          SLIN XP129 WITH $VEL = SVEL_CP(0.1, , LCPDAT33), $TOOL = STOOL2(FP129), $BASE = SBASE(FP129.BASE_NO), $IPO_MODE = SIPO_MODE(FP129.IPO_FRAME), $LOAD = SLOAD(FP129.TOOL_NO), $ACC = SACC_CP(LCPDAT33), $ORI_TYPE = SORI_TYP(LCPDAT33), $APO = SAPO(LCPDAT33), $JERK = SJERK(LCPDAT33), $COLLMON_TOL_PRO[1] = USE_CM_PRO_VALUES(0)
          ;ENDFOLD
          ;FOLD SPTP P500 Vel=100 % PDAT19 Tool[1]:SMC Base[0] ;%{PE}
          ;FOLD Parameters ;%{h}
          ;Params IlfProvider=kukaroboter.basistech.inlineforms.movement.spline; Kuka.IsGlobalPoint=False; Kuka.PointName=P500; Kuka.BlendingEnabled=False; Kuka.MoveDataPtpName=PDAT19; Kuka.VelocityPtp=100; Kuka.VelocityFieldEnabled=True; Kuka.ColDetectFieldEnabled=True; Kuka.CurrentCDSetIndex=0; Kuka.MovementParameterFieldEnabled=True; IlfCommand=SPTP
          ;ENDFOLD
          SPTP XP500 WITH $VEL_AXIS[1] = SVEL_JOINT(100.0), $TOOL = STOOL2(FP500), $BASE = SBASE(FP500.BASE_NO), $IPO_MODE = SIPO_MODE(FP500.IPO_FRAME), $LOAD = SLOAD(FP500.TOOL_NO), $ACC_AXIS[1] = SACC_JOINT(PPDAT19), $APO = SAPO_PTP(PPDAT19), $GEAR_JERK[1] = SGEAR_JERK(PPDAT19), $COLLMON_TOL_PRO[1] = USE_CM_PRO_VALUES(0)
          ;ENDFOLD
          ;FOLD Gripper SET [1]Gripper1 State=[1]ABIERTA Wait 0.2[s] Check with Strategy 1 ;%{PE}
          ;FOLD Parameters Parameters ;%{h}
          ;Params IlfProvider=GripperTech.GripperSet;setgripper=1;setstate=1;setcont=nocont;waittime=0.2;errorstrategy=1
          ;ENDFOLD
          GRPg_SetStateAndCheck(1, 1, 0.2, 1)
          ;ENDFOLD
      ENDIF
      IF eatPosition == 30 THEN
          ;FOLD SPTP P130 Vel=100 % PDAT1 Tool[1]:SMC Base[0] ;%{PE}
          ;FOLD Parameters ;%{h}
          ;Params IlfProvider=kukaroboter.basistech.inlineforms.movement.spline; Kuka.IsGlobalPoint=False; Kuka.PointName=P130; Kuka.BlendingEnabled=False; Kuka.MoveDataPtpName=PDAT1; Kuka.VelocityPtp=100; Kuka.VelocityFieldEnabled=True; Kuka.ColDetectFieldEnabled=True; Kuka.CurrentCDSetIndex=0; Kuka.MovementParameterFieldEnabled=True; IlfCommand=SPTP
          ;ENDFOLD
          SPTP XP130 WITH $VEL_AXIS[1] = SVEL_JOINT(100.0), $TOOL = STOOL2(FP130), $BASE = SBASE(FP130.BASE_NO), $IPO_MODE = SIPO_MODE(FP130.IPO_FRAME), $LOAD = SLOAD(FP130.TOOL_NO), $ACC_AXIS[1] = SACC_JOINT(PPDAT1), $APO = SAPO_PTP(PPDAT1), $GEAR_JERK[1] = SGEAR_JERK(PPDAT1), $COLLMON_TOL_PRO[1] = USE_CM_PRO_VALUES(0)
          ;ENDFOLD
          ;FOLD SLIN P230 Vel=0.1 m/s CPDAT32 Tool[1]:SMC Base[0] ;%{PE}
          ;FOLD Parameters ;%{h}
          ;Params IlfProvider=kukaroboter.basistech.inlineforms.movement.spline; Kuka.IsGlobalPoint=False; Kuka.PointName=P230; Kuka.BlendingEnabled=False; Kuka.MoveDataName=CPDAT32; Kuka.VelocityPath=0.1; Kuka.VelocityFieldEnabled=True; Kuka.ColDetectFieldEnabled=True; Kuka.CurrentCDSetIndex=0; Kuka.MovementParameterFieldEnabled=True; IlfCommand=SLIN
          ;ENDFOLD
          SLIN XP230 WITH $VEL = SVEL_CP(0.1, , LCPDAT32), $TOOL = STOOL2(FP230), $BASE = SBASE(FP230.BASE_NO), $IPO_MODE = SIPO_MODE(FP230.IPO_FRAME), $LOAD = SLOAD(FP230.TOOL_NO), $ACC = SACC_CP(LCPDAT32), $ORI_TYPE = SORI_TYP(LCPDAT32), $APO = SAPO(LCPDAT32), $JERK = SJERK(LCPDAT32), $COLLMON_TOL_PRO[1] = USE_CM_PRO_VALUES(0)
          ;ENDFOLD
          ;FOLD Gripper SET [1]Gripper1 State=[2]CERRADA Wait 0.2[s] Check with Strategy 1 ;%{PE}
          ;FOLD Parameters Parameters ;%{h}
          ;Params IlfProvider=GripperTech.GripperSet;setgripper=1;setstate=2;setcont=nocont;waittime=0.2;errorstrategy=1
          ;ENDFOLD
          GRPg_SetStateAndCheck(1, 2, 0.2, 1)
          ;ENDFOLDinitialPosition
          ;FOLD SLIN P130 Vel=0.1 m/s CPDAT33 Tool[1]:SMC Base[0] ;%{PE}
          ;FOLD Parameters ;%{h}s
          ;Params IlfProvider=kukaroboter.basistech.inlineforms.movement.spline; Kuka.IsGlobalPoint=False; Kuka.PointName=P130; Kuka.BlendingEnabled=False; Kuka.MoveDataName=CPDAT33; Kuka.VelocityPath=0.1; Kuka.VelocityFieldEnabled=True; Kuka.ColDetectFieldEnabled=True; Kuka.CurrentCDSetIndex=0; Kuka.MovementParameterFieldEnabled=True; IlfCommand=SLIN
          ;ENDFOLD
          SLIN XP130 WITH $VEL = SVEL_CP(0.1, , LCPDAT33), $TOOL = STOOL2(FP130), $BASE = SBASE(FP130.BASE_NO), $IPO_MODE = SIPO_MODE(FP130.IPO_FRAME), $LOAD = SLOAD(FP130.TOOL_NO), $ACC = SACC_CP(LCPDAT33), $ORI_TYPE = SORI_TYP(LCPDAT33), $APO = SAPO(LCPDAT33), $JERK = SJERK(LCPDAT33), $COLLMON_TOL_PRO[1] = USE_CM_PRO_VALUES(0)
          ;ENDFOLD
          ;FOLD SPTP P500 Vel=100 % PDAT19 Tool[1]:SMC Base[0] ;%{PE}
          ;FOLD Parameters ;%{h}
          ;Params IlfProvider=kukaroboter.basistech.inlineforms.movement.spline; Kuka.IsGlobalPoint=False; Kuka.PointName=P500; Kuka.BlendingEnabled=False; Kuka.MoveDataPtpName=PDAT19; Kuka.VelocityPtp=100; Kuka.VelocityFieldEnabled=True; Kuka.ColDetectFieldEnabled=True; Kuka.CurrentCDSetIndex=0; Kuka.MovementParameterFieldEnabled=True; IlfCommand=SPTP
          ;ENDFOLD
          SPTP XP500 WITH $VEL_AXIS[1] = SVEL_JOINT(100.0), $TOOL = STOOL2(FP500), $BASE = SBASE(FP500.BASE_NO), $IPO_MODE = SIPO_MODE(FP500.IPO_FRAME), $LOAD = SLOAD(FP500.TOOL_NO), $ACC_AXIS[1] = SACC_JOINT(PPDAT19), $APO = SAPO_PTP(PPDAT19), $GEAR_JERK[1] = SGEAR_JERK(PPDAT19), $COLLMON_TOL_PRO[1] = USE_CM_PRO_VALUES(0)
          ;ENDFOLD
          ;FOLD Gripper SET [1]Gripper1 State=[1]ABIERTA Wait 0.2[s] Check with Strategy 1 ;%{PE}
          ;FOLD Parameters Parameters ;%{h}
          ;Params IlfProvider=GripperTech.GripperSet;setgripper=1;setstate=1;setcont=nocont;waittime=0.2;errorstrategy=1
          ;ENDFOLD
          GRPg_SetStateAndCheck(1, 1, 0.2, 1)
          ;ENDFOLD
      ENDIF
      IF eatPosition == 31 THEN
          ;FOLD SPTP P131 Vel=100 % PDAT1 Tool[1]:SMC Base[0] ;%{PE}
          ;FOLD Parameters ;%{h}
          ;Params IlfProvider=kukaroboter.basistech.inlineforms.movement.spline; Kuka.IsGlobalPoint=False; Kuka.PointName=P131; Kuka.BlendingEnabled=False; Kuka.MoveDataPtpName=PDAT1; Kuka.VelocityPtp=100; Kuka.VelocityFieldEnabled=True; Kuka.ColDetectFieldEnabled=True; Kuka.CurrentCDSetIndex=0; Kuka.MovementParameterFieldEnabled=True; IlfCommand=SPTP
          ;ENDFOLD
          SPTP XP131 WITH $VEL_AXIS[1] = SVEL_JOINT(100.0), $TOOL = STOOL2(FP131), $BASE = SBASE(FP131.BASE_NO), $IPO_MODE = SIPO_MODE(FP131.IPO_FRAME), $LOAD = SLOAD(FP131.TOOL_NO), $ACC_AXIS[1] = SACC_JOINT(PPDAT1), $APO = SAPO_PTP(PPDAT1), $GEAR_JERK[1] = SGEAR_JERK(PPDAT1), $COLLMON_TOL_PRO[1] = USE_CM_PRO_VALUES(0)
          ;ENDFOLD
          ;FOLD SLIN P231 Vel=0.1 m/s CPDAT32 Tool[1]:SMC Base[0] ;%{PE}
          ;FOLD Parameters ;%{h}
          ;Params IlfProvider=kukaroboter.basistech.inlineforms.movement.spline; Kuka.IsGlobalPoint=False; Kuka.PointName=P231; Kuka.BlendingEnabled=False; Kuka.MoveDataName=CPDAT32; Kuka.VelocityPath=0.1; Kuka.VelocityFieldEnabled=True; Kuka.ColDetectFieldEnabled=True; Kuka.CurrentCDSetIndex=0; Kuka.MovementParameterFieldEnabled=True; IlfCommand=SLIN
          ;ENDFOLD
          SLIN XP231 WITH $VEL = SVEL_CP(0.1, , LCPDAT32), $TOOL = STOOL2(FP231), $BASE = SBASE(FP231.BASE_NO), $IPO_MODE = SIPO_MODE(FP231.IPO_FRAME), $LOAD = SLOAD(FP231.TOOL_NO), $ACC = SACC_CP(LCPDAT32), $ORI_TYPE = SORI_TYP(LCPDAT32), $APO = SAPO(LCPDAT32), $JERK = SJERK(LCPDAT32), $COLLMON_TOL_PRO[1] = USE_CM_PRO_VALUES(0)
          ;ENDFOLD
          ;FOLD Gripper SET [1]Gripper1 State=[2]CERRADA Wait 0.2[s] Check with Strategy 1 ;%{PE}
          ;FOLD Parameters Parameters ;%{h}
          ;Params IlfProvider=GripperTech.GripperSet;setgripper=1;setstate=2;setcont=nocont;waittime=0.2;errorstrategy=1
          ;ENDFOLD
          GRPg_SetStateAndCheck(1, 2, 0.2, 1)
          ;ENDFOLDinitialPosition
          ;FOLD SLIN P131 Vel=0.1 m/s CPDAT33 Tool[1]:SMC Base[0] ;%{PE}
          ;FOLD Parameters ;%{h}s
          ;Params IlfProvider=kukaroboter.basistech.inlineforms.movement.spline; Kuka.IsGlobalPoint=False; Kuka.PointName=P131; Kuka.BlendingEnabled=False; Kuka.MoveDataName=CPDAT33; Kuka.VelocityPath=0.1; Kuka.VelocityFieldEnabled=True; Kuka.ColDetectFieldEnabled=True; Kuka.CurrentCDSetIndex=0; Kuka.MovementParameterFieldEnabled=True; IlfCommand=SLIN
          ;ENDFOLD
          SLIN XP131 WITH $VEL = SVEL_CP(0.1, , LCPDAT33), $TOOL = STOOL2(FP131), $BASE = SBASE(FP131.BASE_NO), $IPO_MODE = SIPO_MODE(FP131.IPO_FRAME), $LOAD = SLOAD(FP131.TOOL_NO), $ACC = SACC_CP(LCPDAT33), $ORI_TYPE = SORI_TYP(LCPDAT33), $APO = SAPO(LCPDAT33), $JERK = SJERK(LCPDAT33), $COLLMON_TOL_PRO[1] = USE_CM_PRO_VALUES(0)
          ;ENDFOLD
          ;FOLD SPTP P500 Vel=100 % PDAT19 Tool[1]:SMC Base[0] ;%{PE}
          ;FOLD Parameters ;%{h}
          ;Params IlfProvider=kukaroboter.basistech.inlineforms.movement.spline; Kuka.IsGlobalPoint=False; Kuka.PointName=P500; Kuka.BlendingEnabled=False; Kuka.MoveDataPtpName=PDAT19; Kuka.VelocityPtp=100; Kuka.VelocityFieldEnabled=True; Kuka.ColDetectFieldEnabled=True; Kuka.CurrentCDSetIndex=0; Kuka.MovementParameterFieldEnabled=True; IlfCommand=SPTP
          ;ENDFOLD
          SPTP XP500 WITH $VEL_AXIS[1] = SVEL_JOINT(100.0), $TOOL = STOOL2(FP500), $BASE = SBASE(FP500.BASE_NO), $IPO_MODE = SIPO_MODE(FP500.IPO_FRAME), $LOAD = SLOAD(FP500.TOOL_NO), $ACC_AXIS[1] = SACC_JOINT(PPDAT19), $APO = SAPO_PTP(PPDAT19), $GEAR_JERK[1] = SGEAR_JERK(PPDAT19), $COLLMON_TOL_PRO[1] = USE_CM_PRO_VALUES(0)
          ;ENDFOLD
          ;FOLD Gripper SET [1]Gripper1 State=[1]ABIERTA Wait 0.2[s] Check with Strategy 1 ;%{PE}
          ;FOLD Parameters Parameters ;%{h}
          ;Params IlfProvider=GripperTech.GripperSet;setgripper=1;setstate=1;setcont=nocont;waittime=0.2;errorstrategy=1
          ;ENDFOLD
          GRPg_SetStateAndCheck(1, 1, 0.2, 1)
          ;ENDFOLD
      ENDIF
      IF eatPosition == 32 THEN
          ;FOLD SPTP P132 Vel=100 % PDAT1 Tool[1]:SMC Base[0] ;%{PE}
          ;FOLD Parameters ;%{h}
          ;Params IlfProvider=kukaroboter.basistech.inlineforms.movement.spline; Kuka.IsGlobalPoint=False; Kuka.PointName=P132; Kuka.BlendingEnabled=False; Kuka.MoveDataPtpName=PDAT1; Kuka.VelocityPtp=100; Kuka.VelocityFieldEnabled=True; Kuka.ColDetectFieldEnabled=True; Kuka.CurrentCDSetIndex=0; Kuka.MovementParameterFieldEnabled=True; IlfCommand=SPTP
          ;ENDFOLD
          SPTP XP132 WITH $VEL_AXIS[1] = SVEL_JOINT(100.0), $TOOL = STOOL2(FP132), $BASE = SBASE(FP132.BASE_NO), $IPO_MODE = SIPO_MODE(FP132.IPO_FRAME), $LOAD = SLOAD(FP132.TOOL_NO), $ACC_AXIS[1] = SACC_JOINT(PPDAT1), $APO = SAPO_PTP(PPDAT1), $GEAR_JERK[1] = SGEAR_JERK(PPDAT1), $COLLMON_TOL_PRO[1] = USE_CM_PRO_VALUES(0)
          ;ENDFOLD
          ;FOLD SLIN P232 Vel=0.1 m/s CPDAT32 Tool[1]:SMC Base[0] ;%{PE}
          ;FOLD Parameters ;%{h}
          ;Params IlfProvider=kukaroboter.basistech.inlineforms.movement.spline; Kuka.IsGlobalPoint=False; Kuka.PointName=P232; Kuka.BlendingEnabled=False; Kuka.MoveDataName=CPDAT32; Kuka.VelocityPath=0.1; Kuka.VelocityFieldEnabled=True; Kuka.ColDetectFieldEnabled=True; Kuka.CurrentCDSetIndex=0; Kuka.MovementParameterFieldEnabled=True; IlfCommand=SLIN
          ;ENDFOLD
          SLIN XP232 WITH $VEL = SVEL_CP(0.1, , LCPDAT32), $TOOL = STOOL2(FP232), $BASE = SBASE(FP232.BASE_NO), $IPO_MODE = SIPO_MODE(FP232.IPO_FRAME), $LOAD = SLOAD(FP232.TOOL_NO), $ACC = SACC_CP(LCPDAT32), $ORI_TYPE = SORI_TYP(LCPDAT32), $APO = SAPO(LCPDAT32), $JERK = SJERK(LCPDAT32), $COLLMON_TOL_PRO[1] = USE_CM_PRO_VALUES(0)
          ;ENDFOLD
          ;FOLD Gripper SET [1]Gripper1 State=[2]CERRADA Wait 0.2[s] Check with Strategy 1 ;%{PE}
          ;FOLD Parameters Parameters ;%{h}
          ;Params IlfProvider=GripperTech.GripperSet;setgripper=1;setstate=2;setcont=nocont;waittime=0.2;errorstrategy=1
          ;ENDFOLD
          GRPg_SetStateAndCheck(1, 2, 0.2, 1)
          ;ENDFOLDinitialPosition
          ;FOLD SLIN P132 Vel=0.1 m/s CPDAT33 Tool[1]:SMC Base[0] ;%{PE}
          ;FOLD Parameters ;%{h}s
          ;Params IlfProvider=kukaroboter.basistech.inlineforms.movement.spline; Kuka.IsGlobalPoint=False; Kuka.PointName=P132; Kuka.BlendingEnabled=False; Kuka.MoveDataName=CPDAT33; Kuka.VelocityPath=0.1; Kuka.VelocityFieldEnabled=True; Kuka.ColDetectFieldEnabled=True; Kuka.CurrentCDSetIndex=0; Kuka.MovementParameterFieldEnabled=True; IlfCommand=SLIN
          ;ENDFOLD
          SLIN XP132 WITH $VEL = SVEL_CP(0.1, , LCPDAT33), $TOOL = STOOL2(FP132), $BASE = SBASE(FP132.BASE_NO), $IPO_MODE = SIPO_MODE(FP132.IPO_FRAME), $LOAD = SLOAD(FP132.TOOL_NO), $ACC = SACC_CP(LCPDAT33), $ORI_TYPE = SORI_TYP(LCPDAT33), $APO = SAPO(LCPDAT33), $JERK = SJERK(LCPDAT33), $COLLMON_TOL_PRO[1] = USE_CM_PRO_VALUES(0)
          ;ENDFOLD
          ;FOLD SPTP P500 Vel=100 % PDAT19 Tool[1]:SMC Base[0] ;%{PE}
          ;FOLD Parameters ;%{h}
          ;Params IlfProvider=kukaroboter.basistech.inlineforms.movement.spline; Kuka.IsGlobalPoint=False; Kuka.PointName=P500; Kuka.BlendingEnabled=False; Kuka.MoveDataPtpName=PDAT19; Kuka.VelocityPtp=100; Kuka.VelocityFieldEnabled=True; Kuka.ColDetectFieldEnabled=True; Kuka.CurrentCDSetIndex=0; Kuka.MovementParameterFieldEnabled=True; IlfCommand=SPTP
          ;ENDFOLD
          SPTP XP500 WITH $VEL_AXIS[1] = SVEL_JOINT(100.0), $TOOL = STOOL2(FP500), $BASE = SBASE(FP500.BASE_NO), $IPO_MODE = SIPO_MODE(FP500.IPO_FRAME), $LOAD = SLOAD(FP500.TOOL_NO), $ACC_AXIS[1] = SACC_JOINT(PPDAT19), $APO = SAPO_PTP(PPDAT19), $GEAR_JERK[1] = SGEAR_JERK(PPDAT19), $COLLMON_TOL_PRO[1] = USE_CM_PRO_VALUES(0)
          ;ENDFOLD
          ;FOLD Gripper SET [1]Gripper1 State=[1]ABIERTA Wait 0.2[s] Check with Strategy 1 ;%{PE}
          ;FOLD Parameters Parameters ;%{h}
          ;Params IlfProvider=GripperTech.GripperSet;setgripper=1;setstate=1;setcont=nocont;waittime=0.2;errorstrategy=1
          ;ENDFOLD
          GRPg_SetStateAndCheck(1, 1, 0.2, 1)
          ;ENDFOLD
      ENDIF
      IF eatPosition == 33 THEN
          ;FOLD SPTP P133 Vel=100 % PDAT1 Tool[1]:SMC Base[0] ;%{PE}
          ;FOLD Parameters ;%{h}
          ;Params IlfProvider=kukaroboter.basistech.inlineforms.movement.spline; Kuka.IsGlobalPoint=False; Kuka.PointName=P133; Kuka.BlendingEnabled=False; Kuka.MoveDataPtpName=PDAT1; Kuka.VelocityPtp=100; Kuka.VelocityFieldEnabled=True; Kuka.ColDetectFieldEnabled=True; Kuka.CurrentCDSetIndex=0; Kuka.MovementParameterFieldEnabled=True; IlfCommand=SPTP
          ;ENDFOLD
          SPTP XP133 WITH $VEL_AXIS[1] = SVEL_JOINT(100.0), $TOOL = STOOL2(FP133), $BASE = SBASE(FP133.BASE_NO), $IPO_MODE = SIPO_MODE(FP133.IPO_FRAME), $LOAD = SLOAD(FP133.TOOL_NO), $ACC_AXIS[1] = SACC_JOINT(PPDAT1), $APO = SAPO_PTP(PPDAT1), $GEAR_JERK[1] = SGEAR_JERK(PPDAT1), $COLLMON_TOL_PRO[1] = USE_CM_PRO_VALUES(0)
          ;ENDFOLD
          ;FOLD SLIN P233 Vel=0.1 m/s CPDAT32 Tool[1]:SMC Base[0] ;%{PE}
          ;FOLD Parameters ;%{h}
          ;Params IlfProvider=kukaroboter.basistech.inlineforms.movement.spline; Kuka.IsGlobalPoint=False; Kuka.PointName=P233; Kuka.BlendingEnabled=False; Kuka.MoveDataName=CPDAT32; Kuka.VelocityPath=0.1; Kuka.VelocityFieldEnabled=True; Kuka.ColDetectFieldEnabled=True; Kuka.CurrentCDSetIndex=0; Kuka.MovementParameterFieldEnabled=True; IlfCommand=SLIN
          ;ENDFOLD
          SLIN XP233 WITH $VEL = SVEL_CP(0.1, , LCPDAT32), $TOOL = STOOL2(FP233), $BASE = SBASE(FP233.BASE_NO), $IPO_MODE = SIPO_MODE(FP233.IPO_FRAME), $LOAD = SLOAD(FP233.TOOL_NO), $ACC = SACC_CP(LCPDAT32), $ORI_TYPE = SORI_TYP(LCPDAT32), $APO = SAPO(LCPDAT32), $JERK = SJERK(LCPDAT32), $COLLMON_TOL_PRO[1] = USE_CM_PRO_VALUES(0)
          ;ENDFOLD
          ;FOLD Gripper SET [1]Gripper1 State=[2]CERRADA Wait 0.2[s] Check with Strategy 1 ;%{PE}
          ;FOLD Parameters Parameters ;%{h}
          ;Params IlfProvider=GripperTech.GripperSet;setgripper=1;setstate=2;setcont=nocont;waittime=0.2;errorstrategy=1
          ;ENDFOLD
          GRPg_SetStateAndCheck(1, 2, 0.2, 1)
          ;ENDFOLDinitialPosition
          ;FOLD SLIN P133 Vel=0.1 m/s CPDAT33 Tool[1]:SMC Base[0] ;%{PE}
          ;FOLD Parameters ;%{h}s
          ;Params IlfProvider=kukaroboter.basistech.inlineforms.movement.spline; Kuka.IsGlobalPoint=False; Kuka.PointName=P133; Kuka.BlendingEnabled=False; Kuka.MoveDataName=CPDAT33; Kuka.VelocityPath=0.1; Kuka.VelocityFieldEnabled=True; Kuka.ColDetectFieldEnabled=True; Kuka.CurrentCDSetIndex=0; Kuka.MovementParameterFieldEnabled=True; IlfCommand=SLIN
          ;ENDFOLD
          SLIN XP133 WITH $VEL = SVEL_CP(0.1, , LCPDAT33), $TOOL = STOOL2(FP133), $BASE = SBASE(FP133.BASE_NO), $IPO_MODE = SIPO_MODE(FP133.IPO_FRAME), $LOAD = SLOAD(FP133.TOOL_NO), $ACC = SACC_CP(LCPDAT33), $ORI_TYPE = SORI_TYP(LCPDAT33), $APO = SAPO(LCPDAT33), $JERK = SJERK(LCPDAT33), $COLLMON_TOL_PRO[1] = USE_CM_PRO_VALUES(0)
          ;ENDFOLD
          ;FOLD SPTP P500 Vel=100 % PDAT19 Tool[1]:SMC Base[0] ;%{PE}
          ;FOLD Parameters ;%{h}
          ;Params IlfProvider=kukaroboter.basistech.inlineforms.movement.spline; Kuka.IsGlobalPoint=False; Kuka.PointName=P500; Kuka.BlendingEnabled=False; Kuka.MoveDataPtpName=PDAT19; Kuka.VelocityPtp=100; Kuka.VelocityFieldEnabled=True; Kuka.ColDetectFieldEnabled=True; Kuka.CurrentCDSetIndex=0; Kuka.MovementParameterFieldEnabled=True; IlfCommand=SPTP
          ;ENDFOLD
          SPTP XP500 WITH $VEL_AXIS[1] = SVEL_JOINT(100.0), $TOOL = STOOL2(FP500), $BASE = SBASE(FP500.BASE_NO), $IPO_MODE = SIPO_MODE(FP500.IPO_FRAME), $LOAD = SLOAD(FP500.TOOL_NO), $ACC_AXIS[1] = SACC_JOINT(PPDAT19), $APO = SAPO_PTP(PPDAT19), $GEAR_JERK[1] = SGEAR_JERK(PPDAT19), $COLLMON_TOL_PRO[1] = USE_CM_PRO_VALUES(0)
          ;ENDFOLD
          ;FOLD Gripper SET [1]Gripper1 State=[1]ABIERTA Wait 0.2[s] Check with Strategy 1 ;%{PE}
          ;FOLD Parameters Parameters ;%{h}
          ;Params IlfProvider=GripperTech.GripperSet;setgripper=1;setstate=1;setcont=nocont;waittime=0.2;errorstrategy=1
          ;ENDFOLD
          GRPg_SetStateAndCheck(1, 1, 0.2, 1)
          ;ENDFOLD
      ENDIF
      IF eatPosition == 34 THEN
          ;FOLD SPTP P134 Vel=100 % PDAT1 Tool[1]:SMC Base[0] ;%{PE}
          ;FOLD Parameters ;%{h}
          ;Params IlfProvider=kukaroboter.basistech.inlineforms.movement.spline; Kuka.IsGlobalPoint=False; Kuka.PointName=P134; Kuka.BlendingEnabled=False; Kuka.MoveDataPtpName=PDAT1; Kuka.VelocityPtp=100; Kuka.VelocityFieldEnabled=True; Kuka.ColDetectFieldEnabled=True; Kuka.CurrentCDSetIndex=0; Kuka.MovementParameterFieldEnabled=True; IlfCommand=SPTP
          ;ENDFOLD
          SPTP XP134 WITH $VEL_AXIS[1] = SVEL_JOINT(100.0), $TOOL = STOOL2(FP134), $BASE = SBASE(FP134.BASE_NO), $IPO_MODE = SIPO_MODE(FP134.IPO_FRAME), $LOAD = SLOAD(FP134.TOOL_NO), $ACC_AXIS[1] = SACC_JOINT(PPDAT1), $APO = SAPO_PTP(PPDAT1), $GEAR_JERK[1] = SGEAR_JERK(PPDAT1), $COLLMON_TOL_PRO[1] = USE_CM_PRO_VALUES(0)
          ;ENDFOLD
          ;FOLD SLIN P234 Vel=0.1 m/s CPDAT32 Tool[1]:SMC Base[0] ;%{PE}
          ;FOLD Parameters ;%{h}
          ;Params IlfProvider=kukaroboter.basistech.inlineforms.movement.spline; Kuka.IsGlobalPoint=False; Kuka.PointName=P234; Kuka.BlendingEnabled=False; Kuka.MoveDataName=CPDAT32; Kuka.VelocityPath=0.1; Kuka.VelocityFieldEnabled=True; Kuka.ColDetectFieldEnabled=True; Kuka.CurrentCDSetIndex=0; Kuka.MovementParameterFieldEnabled=True; IlfCommand=SLIN
          ;ENDFOLD
          SLIN XP234 WITH $VEL = SVEL_CP(0.1, , LCPDAT32), $TOOL = STOOL2(FP234), $BASE = SBASE(FP234.BASE_NO), $IPO_MODE = SIPO_MODE(FP234.IPO_FRAME), $LOAD = SLOAD(FP234.TOOL_NO), $ACC = SACC_CP(LCPDAT32), $ORI_TYPE = SORI_TYP(LCPDAT32), $APO = SAPO(LCPDAT32), $JERK = SJERK(LCPDAT32), $COLLMON_TOL_PRO[1] = USE_CM_PRO_VALUES(0)
          ;ENDFOLD
          ;FOLD Gripper SET [1]Gripper1 State=[2]CERRADA Wait 0.2[s] Check with Strategy 1 ;%{PE}
          ;FOLD Parameters Parameters ;%{h}
          ;Params IlfProvider=GripperTech.GripperSet;setgripper=1;setstate=2;setcont=nocont;waittime=0.2;errorstrategy=1
          ;ENDFOLD
          GRPg_SetStateAndCheck(1, 2, 0.2, 1)
          ;ENDFOLDinitialPosition
          ;FOLD SLIN P134 Vel=0.1 m/s CPDAT33 Tool[1]:SMC Base[0] ;%{PE}
          ;FOLD Parameters ;%{h}s
          ;Params IlfProvider=kukaroboter.basistech.inlineforms.movement.spline; Kuka.IsGlobalPoint=False; Kuka.PointName=P134; Kuka.BlendingEnabled=False; Kuka.MoveDataName=CPDAT33; Kuka.VelocityPath=0.1; Kuka.VelocityFieldEnabled=True; Kuka.ColDetectFieldEnabled=True; Kuka.CurrentCDSetIndex=0; Kuka.MovementParameterFieldEnabled=True; IlfCommand=SLIN
          ;ENDFOLD
          SLIN XP134 WITH $VEL = SVEL_CP(0.1, , LCPDAT33), $TOOL = STOOL2(FP134), $BASE = SBASE(FP134.BASE_NO), $IPO_MODE = SIPO_MODE(FP134.IPO_FRAME), $LOAD = SLOAD(FP134.TOOL_NO), $ACC = SACC_CP(LCPDAT33), $ORI_TYPE = SORI_TYP(LCPDAT33), $APO = SAPO(LCPDAT33), $JERK = SJERK(LCPDAT33), $COLLMON_TOL_PRO[1] = USE_CM_PRO_VALUES(0)
          ;ENDFOLD
          ;FOLD SPTP P500 Vel=100 % PDAT19 Tool[1]:SMC Base[0] ;%{PE}
          ;FOLD Parameters ;%{h}
          ;Params IlfProvider=kukaroboter.basistech.inlineforms.movement.spline; Kuka.IsGlobalPoint=False; Kuka.PointName=P500; Kuka.BlendingEnabled=False; Kuka.MoveDataPtpName=PDAT19; Kuka.VelocityPtp=100; Kuka.VelocityFieldEnabled=True; Kuka.ColDetectFieldEnabled=True; Kuka.CurrentCDSetIndex=0; Kuka.MovementParameterFieldEnabled=True; IlfCommand=SPTP
          ;ENDFOLD
          SPTP XP500 WITH $VEL_AXIS[1] = SVEL_JOINT(100.0), $TOOL = STOOL2(FP500), $BASE = SBASE(FP500.BASE_NO), $IPO_MODE = SIPO_MODE(FP500.IPO_FRAME), $LOAD = SLOAD(FP500.TOOL_NO), $ACC_AXIS[1] = SACC_JOINT(PPDAT19), $APO = SAPO_PTP(PPDAT19), $GEAR_JERK[1] = SGEAR_JERK(PPDAT19), $COLLMON_TOL_PRO[1] = USE_CM_PRO_VALUES(0)
          ;ENDFOLD
          ;FOLD Gripper SET [1]Gripper1 State=[1]ABIERTA Wait 0.2[s] Check with Strategy 1 ;%{PE}
          ;FOLD Parameters Parameters ;%{h}
          ;Params IlfProvider=GripperTech.GripperSet;setgripper=1;setstate=1;setcont=nocont;waittime=0.2;errorstrategy=1
          ;ENDFOLD
          GRPg_SetStateAndCheck(1, 1, 0.2, 1)
          ;ENDFOLD
      ENDIF
      IF eatPosition == 35 THEN
          ;FOLD SPTP P135 Vel=100 % PDAT1 Tool[1]:SMC Base[0] ;%{PE}
          ;FOLD Parameters ;%{h}
          ;Params IlfProvider=kukaroboter.basistech.inlineforms.movement.spline; Kuka.IsGlobalPoint=False; Kuka.PointName=P135; Kuka.BlendingEnabled=False; Kuka.MoveDataPtpName=PDAT1; Kuka.VelocityPtp=100; Kuka.VelocityFieldEnabled=True; Kuka.ColDetectFieldEnabled=True; Kuka.CurrentCDSetIndex=0; Kuka.MovementParameterFieldEnabled=True; IlfCommand=SPTP
          ;ENDFOLD
          SPTP XP135 WITH $VEL_AXIS[1] = SVEL_JOINT(100.0), $TOOL = STOOL2(FP135), $BASE = SBASE(FP135.BASE_NO), $IPO_MODE = SIPO_MODE(FP135.IPO_FRAME), $LOAD = SLOAD(FP135.TOOL_NO), $ACC_AXIS[1] = SACC_JOINT(PPDAT1), $APO = SAPO_PTP(PPDAT1), $GEAR_JERK[1] = SGEAR_JERK(PPDAT1), $COLLMON_TOL_PRO[1] = USE_CM_PRO_VALUES(0)
          ;ENDFOLD
          ;FOLD SLIN P235 Vel=0.1 m/s CPDAT32 Tool[1]:SMC Base[0] ;%{PE}
          ;FOLD Parameters ;%{h}
          ;Params IlfProvider=kukaroboter.basistech.inlineforms.movement.spline; Kuka.IsGlobalPoint=False; Kuka.PointName=P235; Kuka.BlendingEnabled=False; Kuka.MoveDataName=CPDAT32; Kuka.VelocityPath=0.1; Kuka.VelocityFieldEnabled=True; Kuka.ColDetectFieldEnabled=True; Kuka.CurrentCDSetIndex=0; Kuka.MovementParameterFieldEnabled=True; IlfCommand=SLIN
          ;ENDFOLD
          SLIN XP235 WITH $VEL = SVEL_CP(0.1, , LCPDAT32), $TOOL = STOOL2(FP235), $BASE = SBASE(FP235.BASE_NO), $IPO_MODE = SIPO_MODE(FP235.IPO_FRAME), $LOAD = SLOAD(FP235.TOOL_NO), $ACC = SACC_CP(LCPDAT32), $ORI_TYPE = SORI_TYP(LCPDAT32), $APO = SAPO(LCPDAT32), $JERK = SJERK(LCPDAT32), $COLLMON_TOL_PRO[1] = USE_CM_PRO_VALUES(0)
          ;ENDFOLD
          ;FOLD Gripper SET [1]Gripper1 State=[2]CERRADA Wait 0.2[s] Check with Strategy 1 ;%{PE}
          ;FOLD Parameters Parameters ;%{h}
          ;Params IlfProvider=GripperTech.GripperSet;setgripper=1;setstate=2;setcont=nocont;waittime=0.2;errorstrategy=1
          ;ENDFOLD
          GRPg_SetStateAndCheck(1, 2, 0.2, 1)
          ;ENDFOLDinitialPosition
          ;FOLD SLIN P135 Vel=0.1 m/s CPDAT33 Tool[1]:SMC Base[0] ;%{PE}
          ;FOLD Parameters ;%{h}s
          ;Params IlfProvider=kukaroboter.basistech.inlineforms.movement.spline; Kuka.IsGlobalPoint=False; Kuka.PointName=P135; Kuka.BlendingEnabled=False; Kuka.MoveDataName=CPDAT33; Kuka.VelocityPath=0.1; Kuka.VelocityFieldEnabled=True; Kuka.ColDetectFieldEnabled=True; Kuka.CurrentCDSetIndex=0; Kuka.MovementParameterFieldEnabled=True; IlfCommand=SLIN
          ;ENDFOLD
          SLIN XP135 WITH $VEL = SVEL_CP(0.1, , LCPDAT33), $TOOL = STOOL2(FP135), $BASE = SBASE(FP135.BASE_NO), $IPO_MODE = SIPO_MODE(FP135.IPO_FRAME), $LOAD = SLOAD(FP135.TOOL_NO), $ACC = SACC_CP(LCPDAT33), $ORI_TYPE = SORI_TYP(LCPDAT33), $APO = SAPO(LCPDAT33), $JERK = SJERK(LCPDAT33), $COLLMON_TOL_PRO[1] = USE_CM_PRO_VALUES(0)
          ;ENDFOLD
          ;FOLD SPTP P500 Vel=100 % PDAT19 Tool[1]:SMC Base[0] ;%{PE}
          ;FOLD Parameters ;%{h}
          ;Params IlfProvider=kukaroboter.basistech.inlineforms.movement.spline; Kuka.IsGlobalPoint=False; Kuka.PointName=P500; Kuka.BlendingEnabled=False; Kuka.MoveDataPtpName=PDAT19; Kuka.VelocityPtp=100; Kuka.VelocityFieldEnabled=True; Kuka.ColDetectFieldEnabled=True; Kuka.CurrentCDSetIndex=0; Kuka.MovementParameterFieldEnabled=True; IlfCommand=SPTP
          ;ENDFOLD
          SPTP XP500 WITH $VEL_AXIS[1] = SVEL_JOINT(100.0), $TOOL = STOOL2(FP500), $BASE = SBASE(FP500.BASE_NO), $IPO_MODE = SIPO_MODE(FP500.IPO_FRAME), $LOAD = SLOAD(FP500.TOOL_NO), $ACC_AXIS[1] = SACC_JOINT(PPDAT19), $APO = SAPO_PTP(PPDAT19), $GEAR_JERK[1] = SGEAR_JERK(PPDAT19), $COLLMON_TOL_PRO[1] = USE_CM_PRO_VALUES(0)
          ;ENDFOLD
          ;FOLD Gripper SET [1]Gripper1 State=[1]ABIERTA Wait 0.2[s] Check with Strategy 1 ;%{PE}
          ;FOLD Parameters Parameters ;%{h}
          ;Params IlfProvider=GripperTech.GripperSet;setgripper=1;setstate=1;setcont=nocont;waittime=0.2;errorstrategy=1
          ;ENDFOLD
          GRPg_SetStateAndCheck(1, 1, 0.2, 1)
          ;ENDFOLD
      ENDIF
      IF eatPosition == 36 THEN
          ;FOLD SPTP P136 Vel=100 % PDAT1 Tool[1]:SMC Base[0] ;%{PE}
          ;FOLD Parameters ;%{h}
          ;Params IlfProvider=kukaroboter.basistech.inlineforms.movement.spline; Kuka.IsGlobalPoint=False; Kuka.PointName=P136; Kuka.BlendingEnabled=False; Kuka.MoveDataPtpName=PDAT1; Kuka.VelocityPtp=100; Kuka.VelocityFieldEnabled=True; Kuka.ColDetectFieldEnabled=True; Kuka.CurrentCDSetIndex=0; Kuka.MovementParameterFieldEnabled=True; IlfCommand=SPTP
          ;ENDFOLD
          SPTP XP136 WITH $VEL_AXIS[1] = SVEL_JOINT(100.0), $TOOL = STOOL2(FP136), $BASE = SBASE(FP136.BASE_NO), $IPO_MODE = SIPO_MODE(FP136.IPO_FRAME), $LOAD = SLOAD(FP136.TOOL_NO), $ACC_AXIS[1] = SACC_JOINT(PPDAT1), $APO = SAPO_PTP(PPDAT1), $GEAR_JERK[1] = SGEAR_JERK(PPDAT1), $COLLMON_TOL_PRO[1] = USE_CM_PRO_VALUES(0)
          ;ENDFOLD
          ;FOLD SLIN P236 Vel=0.1 m/s CPDAT32 Tool[1]:SMC Base[0] ;%{PE}
          ;FOLD Parameters ;%{h}
          ;Params IlfProvider=kukaroboter.basistech.inlineforms.movement.spline; Kuka.IsGlobalPoint=False; Kuka.PointName=P236; Kuka.BlendingEnabled=False; Kuka.MoveDataName=CPDAT32; Kuka.VelocityPath=0.1; Kuka.VelocityFieldEnabled=True; Kuka.ColDetectFieldEnabled=True; Kuka.CurrentCDSetIndex=0; Kuka.MovementParameterFieldEnabled=True; IlfCommand=SLIN
          ;ENDFOLD
          SLIN XP236 WITH $VEL = SVEL_CP(0.1, , LCPDAT32), $TOOL = STOOL2(FP236), $BASE = SBASE(FP236.BASE_NO), $IPO_MODE = SIPO_MODE(FP236.IPO_FRAME), $LOAD = SLOAD(FP236.TOOL_NO), $ACC = SACC_CP(LCPDAT32), $ORI_TYPE = SORI_TYP(LCPDAT32), $APO = SAPO(LCPDAT32), $JERK = SJERK(LCPDAT32), $COLLMON_TOL_PRO[1] = USE_CM_PRO_VALUES(0)
          ;ENDFOLD
          ;FOLD Gripper SET [1]Gripper1 State=[2]CERRADA Wait 0.2[s] Check with Strategy 1 ;%{PE}
          ;FOLD Parameters Parameters ;%{h}
          ;Params IlfProvider=GripperTech.GripperSet;setgripper=1;setstate=2;setcont=nocont;waittime=0.2;errorstrategy=1
          ;ENDFOLD
          GRPg_SetStateAndCheck(1, 2, 0.2, 1)
          ;ENDFOLDinitialPosition
          ;FOLD SLIN P136 Vel=0.1 m/s CPDAT33 Tool[1]:SMC Base[0] ;%{PE}
          ;FOLD Parameters ;%{h}s
          ;Params IlfProvider=kukaroboter.basistech.inlineforms.movement.spline; Kuka.IsGlobalPoint=False; Kuka.PointName=P136; Kuka.BlendingEnabled=False; Kuka.MoveDataName=CPDAT33; Kuka.VelocityPath=0.1; Kuka.VelocityFieldEnabled=True; Kuka.ColDetectFieldEnabled=True; Kuka.CurrentCDSetIndex=0; Kuka.MovementParameterFieldEnabled=True; IlfCommand=SLIN
          ;ENDFOLD
          SLIN XP136 WITH $VEL = SVEL_CP(0.1, , LCPDAT33), $TOOL = STOOL2(FP136), $BASE = SBASE(FP136.BASE_NO), $IPO_MODE = SIPO_MODE(FP136.IPO_FRAME), $LOAD = SLOAD(FP136.TOOL_NO), $ACC = SACC_CP(LCPDAT33), $ORI_TYPE = SORI_TYP(LCPDAT33), $APO = SAPO(LCPDAT33), $JERK = SJERK(LCPDAT33), $COLLMON_TOL_PRO[1] = USE_CM_PRO_VALUES(0)
          ;ENDFOLD
          ;FOLD SPTP P500 Vel=100 % PDAT19 Tool[1]:SMC Base[0] ;%{PE}
          ;FOLD Parameters ;%{h}
          ;Params IlfProvider=kukaroboter.basistech.inlineforms.movement.spline; Kuka.IsGlobalPoint=False; Kuka.PointName=P500; Kuka.BlendingEnabled=False; Kuka.MoveDataPtpName=PDAT19; Kuka.VelocityPtp=100; Kuka.VelocityFieldEnabled=True; Kuka.ColDetectFieldEnabled=True; Kuka.CurrentCDSetIndex=0; Kuka.MovementParameterFieldEnabled=True; IlfCommand=SPTP
          ;ENDFOLD
          SPTP XP500 WITH $VEL_AXIS[1] = SVEL_JOINT(100.0), $TOOL = STOOL2(FP500), $BASE = SBASE(FP500.BASE_NO), $IPO_MODE = SIPO_MODE(FP500.IPO_FRAME), $LOAD = SLOAD(FP500.TOOL_NO), $ACC_AXIS[1] = SACC_JOINT(PPDAT19), $APO = SAPO_PTP(PPDAT19), $GEAR_JERK[1] = SGEAR_JERK(PPDAT19), $COLLMON_TOL_PRO[1] = USE_CM_PRO_VALUES(0)
          ;ENDFOLD
          ;FOLD Gripper SET [1]Gripper1 State=[1]ABIERTA Wait 0.2[s] Check with Strategy 1 ;%{PE}
          ;FOLD Parameters Parameters ;%{h}
          ;Params IlfProvider=GripperTech.GripperSet;setgripper=1;setstate=1;setcont=nocont;waittime=0.2;errorstrategy=1
          ;ENDFOLD
          GRPg_SetStateAndCheck(1, 1, 0.2, 1)
          ;ENDFOLD
      ENDIF
      IF eatPosition == 37 THEN
          ;FOLD SPTP P137 Vel=100 % PDAT1 Tool[1]:SMC Base[0] ;%{PE}
          ;FOLD Parameters ;%{h}
          ;Params IlfProvider=kukaroboter.basistech.inlineforms.movement.spline; Kuka.IsGlobalPoint=False; Kuka.PointName=P137; Kuka.BlendingEnabled=False; Kuka.MoveDataPtpName=PDAT1; Kuka.VelocityPtp=100; Kuka.VelocityFieldEnabled=True; Kuka.ColDetectFieldEnabled=True; Kuka.CurrentCDSetIndex=0; Kuka.MovementParameterFieldEnabled=True; IlfCommand=SPTP
          ;ENDFOLD
          SPTP XP137 WITH $VEL_AXIS[1] = SVEL_JOINT(100.0), $TOOL = STOOL2(FP137), $BASE = SBASE(FP137.BASE_NO), $IPO_MODE = SIPO_MODE(FP137.IPO_FRAME), $LOAD = SLOAD(FP137.TOOL_NO), $ACC_AXIS[1] = SACC_JOINT(PPDAT1), $APO = SAPO_PTP(PPDAT1), $GEAR_JERK[1] = SGEAR_JERK(PPDAT1), $COLLMON_TOL_PRO[1] = USE_CM_PRO_VALUES(0)
          ;ENDFOLD
          ;FOLD SLIN P237 Vel=0.1 m/s CPDAT32 Tool[1]:SMC Base[0] ;%{PE}
          ;FOLD Parameters ;%{h}
          ;Params IlfProvider=kukaroboter.basistech.inlineforms.movement.spline; Kuka.IsGlobalPoint=False; Kuka.PointName=P237; Kuka.BlendingEnabled=False; Kuka.MoveDataName=CPDAT32; Kuka.VelocityPath=0.1; Kuka.VelocityFieldEnabled=True; Kuka.ColDetectFieldEnabled=True; Kuka.CurrentCDSetIndex=0; Kuka.MovementParameterFieldEnabled=True; IlfCommand=SLIN
          ;ENDFOLD
          SLIN XP237 WITH $VEL = SVEL_CP(0.1, , LCPDAT32), $TOOL = STOOL2(FP237), $BASE = SBASE(FP237.BASE_NO), $IPO_MODE = SIPO_MODE(FP237.IPO_FRAME), $LOAD = SLOAD(FP237.TOOL_NO), $ACC = SACC_CP(LCPDAT32), $ORI_TYPE = SORI_TYP(LCPDAT32), $APO = SAPO(LCPDAT32), $JERK = SJERK(LCPDAT32), $COLLMON_TOL_PRO[1] = USE_CM_PRO_VALUES(0)
          ;ENDFOLD
          ;FOLD Gripper SET [1]Gripper1 State=[2]CERRADA Wait 0.2[s] Check with Strategy 1 ;%{PE}
          ;FOLD Parameters Parameters ;%{h}
          ;Params IlfProvider=GripperTech.GripperSet;setgripper=1;setstate=2;setcont=nocont;waittime=0.2;errorstrategy=1
          ;ENDFOLD
          GRPg_SetStateAndCheck(1, 2, 0.2, 1)
          ;ENDFOLDinitialPosition
          ;FOLD SLIN P137 Vel=0.1 m/s CPDAT33 Tool[1]:SMC Base[0] ;%{PE}
          ;FOLD Parameters ;%{h}s
          ;Params IlfProvider=kukaroboter.basistech.inlineforms.movement.spline; Kuka.IsGlobalPoint=False; Kuka.PointName=P137; Kuka.BlendingEnabled=False; Kuka.MoveDataName=CPDAT33; Kuka.VelocityPath=0.1; Kuka.VelocityFieldEnabled=True; Kuka.ColDetectFieldEnabled=True; Kuka.CurrentCDSetIndex=0; Kuka.MovementParameterFieldEnabled=True; IlfCommand=SLIN
          ;ENDFOLD
          SLIN XP137 WITH $VEL = SVEL_CP(0.1, , LCPDAT33), $TOOL = STOOL2(FP137), $BASE = SBASE(FP137.BASE_NO), $IPO_MODE = SIPO_MODE(FP137.IPO_FRAME), $LOAD = SLOAD(FP137.TOOL_NO), $ACC = SACC_CP(LCPDAT33), $ORI_TYPE = SORI_TYP(LCPDAT33), $APO = SAPO(LCPDAT33), $JERK = SJERK(LCPDAT33), $COLLMON_TOL_PRO[1] = USE_CM_PRO_VALUES(0)
          ;ENDFOLD
          ;FOLD SPTP P500 Vel=100 % PDAT19 Tool[1]:SMC Base[0] ;%{PE}
          ;FOLD Parameters ;%{h}
          ;Params IlfProvider=kukaroboter.basistech.inlineforms.movement.spline; Kuka.IsGlobalPoint=False; Kuka.PointName=P500; Kuka.BlendingEnabled=False; Kuka.MoveDataPtpName=PDAT19; Kuka.VelocityPtp=100; Kuka.VelocityFieldEnabled=True; Kuka.ColDetectFieldEnabled=True; Kuka.CurrentCDSetIndex=0; Kuka.MovementParameterFieldEnabled=True; IlfCommand=SPTP
          ;ENDFOLD
          SPTP XP500 WITH $VEL_AXIS[1] = SVEL_JOINT(100.0), $TOOL = STOOL2(FP500), $BASE = SBASE(FP500.BASE_NO), $IPO_MODE = SIPO_MODE(FP500.IPO_FRAME), $LOAD = SLOAD(FP500.TOOL_NO), $ACC_AXIS[1] = SACC_JOINT(PPDAT19), $APO = SAPO_PTP(PPDAT19), $GEAR_JERK[1] = SGEAR_JERK(PPDAT19), $COLLMON_TOL_PRO[1] = USE_CM_PRO_VALUES(0)
          ;ENDFOLD
          ;FOLD Gripper SET [1]Gripper1 State=[1]ABIERTA Wait 0.2[s] Check with Strategy 1 ;%{PE}
          ;FOLD Parameters Parameters ;%{h}
          ;Params IlfProvider=GripperTech.GripperSet;setgripper=1;setstate=1;setcont=nocont;waittime=0.2;errorstrategy=1
          ;ENDFOLD
          GRPg_SetStateAndCheck(1, 1, 0.2, 1)
          ;ENDFOLD
      ENDIF
      IF eatPosition == 38 THEN
          ;FOLD SPTP P138 Vel=100 % PDAT1 Tool[1]:SMC Base[0] ;%{PE}
          ;FOLD Parameters ;%{h}
          ;Params IlfProvider=kukaroboter.basistech.inlineforms.movement.spline; Kuka.IsGlobalPoint=False; Kuka.PointName=P138; Kuka.BlendingEnabled=False; Kuka.MoveDataPtpName=PDAT1; Kuka.VelocityPtp=100; Kuka.VelocityFieldEnabled=True; Kuka.ColDetectFieldEnabled=True; Kuka.CurrentCDSetIndex=0; Kuka.MovementParameterFieldEnabled=True; IlfCommand=SPTP
          ;ENDFOLD
          SPTP XP138 WITH $VEL_AXIS[1] = SVEL_JOINT(100.0), $TOOL = STOOL2(FP138), $BASE = SBASE(FP138.BASE_NO), $IPO_MODE = SIPO_MODE(FP138.IPO_FRAME), $LOAD = SLOAD(FP138.TOOL_NO), $ACC_AXIS[1] = SACC_JOINT(PPDAT1), $APO = SAPO_PTP(PPDAT1), $GEAR_JERK[1] = SGEAR_JERK(PPDAT1), $COLLMON_TOL_PRO[1] = USE_CM_PRO_VALUES(0)
          ;ENDFOLD
          ;FOLD SLIN P238 Vel=0.1 m/s CPDAT32 Tool[1]:SMC Base[0] ;%{PE}
          ;FOLD Parameters ;%{h}
          ;Params IlfProvider=kukaroboter.basistech.inlineforms.movement.spline; Kuka.IsGlobalPoint=False; Kuka.PointName=P238; Kuka.BlendingEnabled=False; Kuka.MoveDataName=CPDAT32; Kuka.VelocityPath=0.1; Kuka.VelocityFieldEnabled=True; Kuka.ColDetectFieldEnabled=True; Kuka.CurrentCDSetIndex=0; Kuka.MovementParameterFieldEnabled=True; IlfCommand=SLIN
          ;ENDFOLD
          SLIN XP238 WITH $VEL = SVEL_CP(0.1, , LCPDAT32), $TOOL = STOOL2(FP238), $BASE = SBASE(FP238.BASE_NO), $IPO_MODE = SIPO_MODE(FP238.IPO_FRAME), $LOAD = SLOAD(FP238.TOOL_NO), $ACC = SACC_CP(LCPDAT32), $ORI_TYPE = SORI_TYP(LCPDAT32), $APO = SAPO(LCPDAT32), $JERK = SJERK(LCPDAT32), $COLLMON_TOL_PRO[1] = USE_CM_PRO_VALUES(0)
          ;ENDFOLD
          ;FOLD Gripper SET [1]Gripper1 State=[2]CERRADA Wait 0.2[s] Check with Strategy 1 ;%{PE}
          ;FOLD Parameters Parameters ;%{h}
          ;Params IlfProvider=GripperTech.GripperSet;setgripper=1;setstate=2;setcont=nocont;waittime=0.2;errorstrategy=1
          ;ENDFOLD
          GRPg_SetStateAndCheck(1, 2, 0.2, 1)
          ;ENDFOLDinitialPosition
          ;FOLD SLIN P138 Vel=0.1 m/s CPDAT33 Tool[1]:SMC Base[0] ;%{PE}
          ;FOLD Parameters ;%{h}s
          ;Params IlfProvider=kukaroboter.basistech.inlineforms.movement.spline; Kuka.IsGlobalPoint=False; Kuka.PointName=P138; Kuka.BlendingEnabled=False; Kuka.MoveDataName=CPDAT33; Kuka.VelocityPath=0.1; Kuka.VelocityFieldEnabled=True; Kuka.ColDetectFieldEnabled=True; Kuka.CurrentCDSetIndex=0; Kuka.MovementParameterFieldEnabled=True; IlfCommand=SLIN
          ;ENDFOLD
          SLIN XP138 WITH $VEL = SVEL_CP(0.1, , LCPDAT33), $TOOL = STOOL2(FP138), $BASE = SBASE(FP138.BASE_NO), $IPO_MODE = SIPO_MODE(FP138.IPO_FRAME), $LOAD = SLOAD(FP138.TOOL_NO), $ACC = SACC_CP(LCPDAT33), $ORI_TYPE = SORI_TYP(LCPDAT33), $APO = SAPO(LCPDAT33), $JERK = SJERK(LCPDAT33), $COLLMON_TOL_PRO[1] = USE_CM_PRO_VALUES(0)
          ;ENDFOLD
          ;FOLD SPTP P500 Vel=100 % PDAT19 Tool[1]:SMC Base[0] ;%{PE}
          ;FOLD Parameters ;%{h}
          ;Params IlfProvider=kukaroboter.basistech.inlineforms.movement.spline; Kuka.IsGlobalPoint=False; Kuka.PointName=P500; Kuka.BlendingEnabled=False; Kuka.MoveDataPtpName=PDAT19; Kuka.VelocityPtp=100; Kuka.VelocityFieldEnabled=True; Kuka.ColDetectFieldEnabled=True; Kuka.CurrentCDSetIndex=0; Kuka.MovementParameterFieldEnabled=True; IlfCommand=SPTP
          ;ENDFOLD
          SPTP XP500 WITH $VEL_AXIS[1] = SVEL_JOINT(100.0), $TOOL = STOOL2(FP500), $BASE = SBASE(FP500.BASE_NO), $IPO_MODE = SIPO_MODE(FP500.IPO_FRAME), $LOAD = SLOAD(FP500.TOOL_NO), $ACC_AXIS[1] = SACC_JOINT(PPDAT19), $APO = SAPO_PTP(PPDAT19), $GEAR_JERK[1] = SGEAR_JERK(PPDAT19), $COLLMON_TOL_PRO[1] = USE_CM_PRO_VALUES(0)
          ;ENDFOLD
          ;FOLD Gripper SET [1]Gripper1 State=[1]ABIERTA Wait 0.2[s] Check with Strategy 1 ;%{PE}
          ;FOLD Parameters Parameters ;%{h}
          ;Params IlfProvider=GripperTech.GripperSet;setgripper=1;setstate=1;setcont=nocont;waittime=0.2;errorstrategy=1
          ;ENDFOLD
          GRPg_SetStateAndCheck(1, 1, 0.2, 1)
          ;ENDFOLD
      ENDIF
      IF eatPosition == 39 THEN
          ;FOLD SPTP P139 Vel=100 % PDAT1 Tool[1]:SMC Base[0] ;%{PE}
          ;FOLD Parameters ;%{h}
          ;Params IlfProvider=kukaroboter.basistech.inlineforms.movement.spline; Kuka.IsGlobalPoint=False; Kuka.PointName=P139; Kuka.BlendingEnabled=False; Kuka.MoveDataPtpName=PDAT1; Kuka.VelocityPtp=100; Kuka.VelocityFieldEnabled=True; Kuka.ColDetectFieldEnabled=True; Kuka.CurrentCDSetIndex=0; Kuka.MovementParameterFieldEnabled=True; IlfCommand=SPTP
          ;ENDFOLD
          SPTP XP139 WITH $VEL_AXIS[1] = SVEL_JOINT(100.0), $TOOL = STOOL2(FP139), $BASE = SBASE(FP139.BASE_NO), $IPO_MODE = SIPO_MODE(FP139.IPO_FRAME), $LOAD = SLOAD(FP139.TOOL_NO), $ACC_AXIS[1] = SACC_JOINT(PPDAT1), $APO = SAPO_PTP(PPDAT1), $GEAR_JERK[1] = SGEAR_JERK(PPDAT1), $COLLMON_TOL_PRO[1] = USE_CM_PRO_VALUES(0)
          ;ENDFOLD
          ;FOLD SLIN P239 Vel=0.1 m/s CPDAT32 Tool[1]:SMC Base[0] ;%{PE}
          ;FOLD Parameters ;%{h}
          ;Params IlfProvider=kukaroboter.basistech.inlineforms.movement.spline; Kuka.IsGlobalPoint=False; Kuka.PointName=P239; Kuka.BlendingEnabled=False; Kuka.MoveDataName=CPDAT32; Kuka.VelocityPath=0.1; Kuka.VelocityFieldEnabled=True; Kuka.ColDetectFieldEnabled=True; Kuka.CurrentCDSetIndex=0; Kuka.MovementParameterFieldEnabled=True; IlfCommand=SLIN
          ;ENDFOLD
          SLIN XP239 WITH $VEL = SVEL_CP(0.1, , LCPDAT32), $TOOL = STOOL2(FP239), $BASE = SBASE(FP239.BASE_NO), $IPO_MODE = SIPO_MODE(FP239.IPO_FRAME), $LOAD = SLOAD(FP239.TOOL_NO), $ACC = SACC_CP(LCPDAT32), $ORI_TYPE = SORI_TYP(LCPDAT32), $APO = SAPO(LCPDAT32), $JERK = SJERK(LCPDAT32), $COLLMON_TOL_PRO[1] = USE_CM_PRO_VALUES(0)
          ;ENDFOLD
          ;FOLD Gripper SET [1]Gripper1 State=[2]CERRADA Wait 0.2[s] Check with Strategy 1 ;%{PE}
          ;FOLD Parameters Parameters ;%{h}
          ;Params IlfProvider=GripperTech.GripperSet;setgripper=1;setstate=2;setcont=nocont;waittime=0.2;errorstrategy=1
          ;ENDFOLD
          GRPg_SetStateAndCheck(1, 2, 0.2, 1)
          ;ENDFOLDinitialPosition
          ;FOLD SLIN P139 Vel=0.1 m/s CPDAT33 Tool[1]:SMC Base[0] ;%{PE}
          ;FOLD Parameters ;%{h}s
          ;Params IlfProvider=kukaroboter.basistech.inlineforms.movement.spline; Kuka.IsGlobalPoint=False; Kuka.PointName=P139; Kuka.BlendingEnabled=False; Kuka.MoveDataName=CPDAT33; Kuka.VelocityPath=0.1; Kuka.VelocityFieldEnabled=True; Kuka.ColDetectFieldEnabled=True; Kuka.CurrentCDSetIndex=0; Kuka.MovementParameterFieldEnabled=True; IlfCommand=SLIN
          ;ENDFOLD
          SLIN XP139 WITH $VEL = SVEL_CP(0.1, , LCPDAT33), $TOOL = STOOL2(FP139), $BASE = SBASE(FP139.BASE_NO), $IPO_MODE = SIPO_MODE(FP139.IPO_FRAME), $LOAD = SLOAD(FP139.TOOL_NO), $ACC = SACC_CP(LCPDAT33), $ORI_TYPE = SORI_TYP(LCPDAT33), $APO = SAPO(LCPDAT33), $JERK = SJERK(LCPDAT33), $COLLMON_TOL_PRO[1] = USE_CM_PRO_VALUES(0)
          ;ENDFOLD
          ;FOLD SPTP P500 Vel=100 % PDAT19 Tool[1]:SMC Base[0] ;%{PE}
          ;FOLD Parameters ;%{h}
          ;Params IlfProvider=kukaroboter.basistech.inlineforms.movement.spline; Kuka.IsGlobalPoint=False; Kuka.PointName=P500; Kuka.BlendingEnabled=False; Kuka.MoveDataPtpName=PDAT19; Kuka.VelocityPtp=100; Kuka.VelocityFieldEnabled=True; Kuka.ColDetectFieldEnabled=True; Kuka.CurrentCDSetIndex=0; Kuka.MovementParameterFieldEnabled=True; IlfCommand=SPTP
          ;ENDFOLD
          SPTP XP500 WITH $VEL_AXIS[1] = SVEL_JOINT(100.0), $TOOL = STOOL2(FP500), $BASE = SBASE(FP500.BASE_NO), $IPO_MODE = SIPO_MODE(FP500.IPO_FRAME), $LOAD = SLOAD(FP500.TOOL_NO), $ACC_AXIS[1] = SACC_JOINT(PPDAT19), $APO = SAPO_PTP(PPDAT19), $GEAR_JERK[1] = SGEAR_JERK(PPDAT19), $COLLMON_TOL_PRO[1] = USE_CM_PRO_VALUES(0)
          ;ENDFOLD
          ;FOLD Gripper SET [1]Gripper1 State=[1]ABIERTA Wait 0.2[s] Check with Strategy 1 ;%{PE}
          ;FOLD Parameters Parameters ;%{h}
          ;Params IlfProvider=GripperTech.GripperSet;setgripper=1;setstate=1;setcont=nocont;waittime=0.2;errorstrategy=1
          ;ENDFOLD
          GRPg_SetStateAndCheck(1, 1, 0.2, 1)
          ;ENDFOLD
      ENDIF
      IF eatPosition == 40 THEN
          ;FOLD SPTP P140 Vel=100 % PDAT1 Tool[1]:SMC Base[0] ;%{PE}
          ;FOLD Parameters ;%{h}
          ;Params IlfProvider=kukaroboter.basistech.inlineforms.movement.spline; Kuka.IsGlobalPoint=False; Kuka.PointName=P140; Kuka.BlendingEnabled=False; Kuka.MoveDataPtpName=PDAT1; Kuka.VelocityPtp=100; Kuka.VelocityFieldEnabled=True; Kuka.ColDetectFieldEnabled=True; Kuka.CurrentCDSetIndex=0; Kuka.MovementParameterFieldEnabled=True; IlfCommand=SPTP
          ;ENDFOLD
          SPTP XP140 WITH $VEL_AXIS[1] = SVEL_JOINT(100.0), $TOOL = STOOL2(FP140), $BASE = SBASE(FP140.BASE_NO), $IPO_MODE = SIPO_MODE(FP140.IPO_FRAME), $LOAD = SLOAD(FP140.TOOL_NO), $ACC_AXIS[1] = SACC_JOINT(PPDAT1), $APO = SAPO_PTP(PPDAT1), $GEAR_JERK[1] = SGEAR_JERK(PPDAT1), $COLLMON_TOL_PRO[1] = USE_CM_PRO_VALUES(0)
          ;ENDFOLD
          ;FOLD SLIN P240 Vel=0.1 m/s CPDAT32 Tool[1]:SMC Base[0] ;%{PE}
          ;FOLD Parameters ;%{h}
          ;Params IlfProvider=kukaroboter.basistech.inlineforms.movement.spline; Kuka.IsGlobalPoint=False; Kuka.PointName=P240; Kuka.BlendingEnabled=False; Kuka.MoveDataName=CPDAT32; Kuka.VelocityPath=0.1; Kuka.VelocityFieldEnabled=True; Kuka.ColDetectFieldEnabled=True; Kuka.CurrentCDSetIndex=0; Kuka.MovementParameterFieldEnabled=True; IlfCommand=SLIN
          ;ENDFOLD
          SLIN XP240 WITH $VEL = SVEL_CP(0.1, , LCPDAT32), $TOOL = STOOL2(FP240), $BASE = SBASE(FP240.BASE_NO), $IPO_MODE = SIPO_MODE(FP240.IPO_FRAME), $LOAD = SLOAD(FP240.TOOL_NO), $ACC = SACC_CP(LCPDAT32), $ORI_TYPE = SORI_TYP(LCPDAT32), $APO = SAPO(LCPDAT32), $JERK = SJERK(LCPDAT32), $COLLMON_TOL_PRO[1] = USE_CM_PRO_VALUES(0)
          ;ENDFOLD
          ;FOLD Gripper SET [1]Gripper1 State=[2]CERRADA Wait 0.2[s] Check with Strategy 1 ;%{PE}
          ;FOLD Parameters Parameters ;%{h}
          ;Params IlfProvider=GripperTech.GripperSet;setgripper=1;setstate=2;setcont=nocont;waittime=0.2;errorstrategy=1
          ;ENDFOLD
          GRPg_SetStateAndCheck(1, 2, 0.2, 1)
          ;ENDFOLDinitialPosition
          ;FOLD SLIN P140 Vel=0.1 m/s CPDAT33 Tool[1]:SMC Base[0] ;%{PE}
          ;FOLD Parameters ;%{h}s
          ;Params IlfProvider=kukaroboter.basistech.inlineforms.movement.spline; Kuka.IsGlobalPoint=False; Kuka.PointName=P140; Kuka.BlendingEnabled=False; Kuka.MoveDataName=CPDAT33; Kuka.VelocityPath=0.1; Kuka.VelocityFieldEnabled=True; Kuka.ColDetectFieldEnabled=True; Kuka.CurrentCDSetIndex=0; Kuka.MovementParameterFieldEnabled=True; IlfCommand=SLIN
          ;ENDFOLD
          SLIN XP140 WITH $VEL = SVEL_CP(0.1, , LCPDAT33), $TOOL = STOOL2(FP140), $BASE = SBASE(FP140.BASE_NO), $IPO_MODE = SIPO_MODE(FP140.IPO_FRAME), $LOAD = SLOAD(FP140.TOOL_NO), $ACC = SACC_CP(LCPDAT33), $ORI_TYPE = SORI_TYP(LCPDAT33), $APO = SAPO(LCPDAT33), $JERK = SJERK(LCPDAT33), $COLLMON_TOL_PRO[1] = USE_CM_PRO_VALUES(0)
          ;ENDFOLD
          ;FOLD SPTP P500 Vel=100 % PDAT19 Tool[1]:SMC Base[0] ;%{PE}
          ;FOLD Parameters ;%{h}
          ;Params IlfProvider=kukaroboter.basistech.inlineforms.movement.spline; Kuka.IsGlobalPoint=False; Kuka.PointName=P500; Kuka.BlendingEnabled=False; Kuka.MoveDataPtpName=PDAT19; Kuka.VelocityPtp=100; Kuka.VelocityFieldEnabled=True; Kuka.ColDetectFieldEnabled=True; Kuka.CurrentCDSetIndex=0; Kuka.MovementParameterFieldEnabled=True; IlfCommand=SPTP
          ;ENDFOLD
          SPTP XP500 WITH $VEL_AXIS[1] = SVEL_JOINT(100.0), $TOOL = STOOL2(FP500), $BASE = SBASE(FP500.BASE_NO), $IPO_MODE = SIPO_MODE(FP500.IPO_FRAME), $LOAD = SLOAD(FP500.TOOL_NO), $ACC_AXIS[1] = SACC_JOINT(PPDAT19), $APO = SAPO_PTP(PPDAT19), $GEAR_JERK[1] = SGEAR_JERK(PPDAT19), $COLLMON_TOL_PRO[1] = USE_CM_PRO_VALUES(0)
          ;ENDFOLD
          ;FOLD Gripper SET [1]Gripper1 State=[1]ABIERTA Wait 0.2[s] Check with Strategy 1 ;%{PE}
          ;FOLD Parameters Parameters ;%{h}
          ;Params IlfProvider=GripperTech.GripperSet;setgripper=1;setstate=1;setcont=nocont;waittime=0.2;errorstrategy=1
          ;ENDFOLD
          GRPg_SetStateAndCheck(1, 1, 0.2, 1)
          ;ENDFOLD
      ENDIF
      IF eatPosition == 41 THEN
          ;FOLD SPTP P141 Vel=100 % PDAT1 Tool[1]:SMC Base[0] ;%{PE}
          ;FOLD Parameters ;%{h}
          ;Params IlfProvider=kukaroboter.basistech.inlineforms.movement.spline; Kuka.IsGlobalPoint=False; Kuka.PointName=P141; Kuka.BlendingEnabled=False; Kuka.MoveDataPtpName=PDAT1; Kuka.VelocityPtp=100; Kuka.VelocityFieldEnabled=True; Kuka.ColDetectFieldEnabled=True; Kuka.CurrentCDSetIndex=0; Kuka.MovementParameterFieldEnabled=True; IlfCommand=SPTP
          ;ENDFOLD
          SPTP XP141 WITH $VEL_AXIS[1] = SVEL_JOINT(100.0), $TOOL = STOOL2(FP141), $BASE = SBASE(FP141.BASE_NO), $IPO_MODE = SIPO_MODE(FP141.IPO_FRAME), $LOAD = SLOAD(FP141.TOOL_NO), $ACC_AXIS[1] = SACC_JOINT(PPDAT1), $APO = SAPO_PTP(PPDAT1), $GEAR_JERK[1] = SGEAR_JERK(PPDAT1), $COLLMON_TOL_PRO[1] = USE_CM_PRO_VALUES(0)
          ;ENDFOLD
          ;FOLD SLIN P241 Vel=0.1 m/s CPDAT32 Tool[1]:SMC Base[0] ;%{PE}
          ;FOLD Parameters ;%{h}
          ;Params IlfProvider=kukaroboter.basistech.inlineforms.movement.spline; Kuka.IsGlobalPoint=False; Kuka.PointName=P241; Kuka.BlendingEnabled=False; Kuka.MoveDataName=CPDAT32; Kuka.VelocityPath=0.1; Kuka.VelocityFieldEnabled=True; Kuka.ColDetectFieldEnabled=True; Kuka.CurrentCDSetIndex=0; Kuka.MovementParameterFieldEnabled=True; IlfCommand=SLIN
          ;ENDFOLD
          SLIN XP241 WITH $VEL = SVEL_CP(0.1, , LCPDAT32), $TOOL = STOOL2(FP241), $BASE = SBASE(FP241.BASE_NO), $IPO_MODE = SIPO_MODE(FP241.IPO_FRAME), $LOAD = SLOAD(FP241.TOOL_NO), $ACC = SACC_CP(LCPDAT32), $ORI_TYPE = SORI_TYP(LCPDAT32), $APO = SAPO(LCPDAT32), $JERK = SJERK(LCPDAT32), $COLLMON_TOL_PRO[1] = USE_CM_PRO_VALUES(0)
          ;ENDFOLD
          ;FOLD Gripper SET [1]Gripper1 State=[2]CERRADA Wait 0.2[s] Check with Strategy 1 ;%{PE}
          ;FOLD Parameters Parameters ;%{h}
          ;Params IlfProvider=GripperTech.GripperSet;setgripper=1;setstate=2;setcont=nocont;waittime=0.2;errorstrategy=1
          ;ENDFOLD
          GRPg_SetStateAndCheck(1, 2, 0.2, 1)
          ;ENDFOLDinitialPosition
          ;FOLD SLIN P141 Vel=0.1 m/s CPDAT33 Tool[1]:SMC Base[0] ;%{PE}
          ;FOLD Parameters ;%{h}s
          ;Params IlfProvider=kukaroboter.basistech.inlineforms.movement.spline; Kuka.IsGlobalPoint=False; Kuka.PointName=P141; Kuka.BlendingEnabled=False; Kuka.MoveDataName=CPDAT33; Kuka.VelocityPath=0.1; Kuka.VelocityFieldEnabled=True; Kuka.ColDetectFieldEnabled=True; Kuka.CurrentCDSetIndex=0; Kuka.MovementParameterFieldEnabled=True; IlfCommand=SLIN
          ;ENDFOLD
          SLIN XP141 WITH $VEL = SVEL_CP(0.1, , LCPDAT33), $TOOL = STOOL2(FP141), $BASE = SBASE(FP141.BASE_NO), $IPO_MODE = SIPO_MODE(FP141.IPO_FRAME), $LOAD = SLOAD(FP141.TOOL_NO), $ACC = SACC_CP(LCPDAT33), $ORI_TYPE = SORI_TYP(LCPDAT33), $APO = SAPO(LCPDAT33), $JERK = SJERK(LCPDAT33), $COLLMON_TOL_PRO[1] = USE_CM_PRO_VALUES(0)
          ;ENDFOLD
          ;FOLD SPTP P500 Vel=100 % PDAT19 Tool[1]:SMC Base[0] ;%{PE}
          ;FOLD Parameters ;%{h}
          ;Params IlfProvider=kukaroboter.basistech.inlineforms.movement.spline; Kuka.IsGlobalPoint=False; Kuka.PointName=P500; Kuka.BlendingEnabled=False; Kuka.MoveDataPtpName=PDAT19; Kuka.VelocityPtp=100; Kuka.VelocityFieldEnabled=True; Kuka.ColDetectFieldEnabled=True; Kuka.CurrentCDSetIndex=0; Kuka.MovementParameterFieldEnabled=True; IlfCommand=SPTP
          ;ENDFOLD
          SPTP XP500 WITH $VEL_AXIS[1] = SVEL_JOINT(100.0), $TOOL = STOOL2(FP500), $BASE = SBASE(FP500.BASE_NO), $IPO_MODE = SIPO_MODE(FP500.IPO_FRAME), $LOAD = SLOAD(FP500.TOOL_NO), $ACC_AXIS[1] = SACC_JOINT(PPDAT19), $APO = SAPO_PTP(PPDAT19), $GEAR_JERK[1] = SGEAR_JERK(PPDAT19), $COLLMON_TOL_PRO[1] = USE_CM_PRO_VALUES(0)
          ;ENDFOLD
          ;FOLD Gripper SET [1]Gripper1 State=[1]ABIERTA Wait 0.2[s] Check with Strategy 1 ;%{PE}
          ;FOLD Parameters Parameters ;%{h}
          ;Params IlfProvider=GripperTech.GripperSet;setgripper=1;setstate=1;setcont=nocont;waittime=0.2;errorstrategy=1
          ;ENDFOLD
          GRPg_SetStateAndCheck(1, 1, 0.2, 1)
          ;ENDFOLD
      ENDIF
      IF eatPosition == 42 THEN
          ;FOLD SPTP P142 Vel=100 % PDAT1 Tool[1]:SMC Base[0] ;%{PE}
          ;FOLD Parameters ;%{h}
          ;Params IlfProvider=kukaroboter.basistech.inlineforms.movement.spline; Kuka.IsGlobalPoint=False; Kuka.PointName=P142; Kuka.BlendingEnabled=False; Kuka.MoveDataPtpName=PDAT1; Kuka.VelocityPtp=100; Kuka.VelocityFieldEnabled=True; Kuka.ColDetectFieldEnabled=True; Kuka.CurrentCDSetIndex=0; Kuka.MovementParameterFieldEnabled=True; IlfCommand=SPTP
          ;ENDFOLD
          SPTP XP142 WITH $VEL_AXIS[1] = SVEL_JOINT(100.0), $TOOL = STOOL2(FP142), $BASE = SBASE(FP142.BASE_NO), $IPO_MODE = SIPO_MODE(FP142.IPO_FRAME), $LOAD = SLOAD(FP142.TOOL_NO), $ACC_AXIS[1] = SACC_JOINT(PPDAT1), $APO = SAPO_PTP(PPDAT1), $GEAR_JERK[1] = SGEAR_JERK(PPDAT1), $COLLMON_TOL_PRO[1] = USE_CM_PRO_VALUES(0)
          ;ENDFOLD
          ;FOLD SLIN P242 Vel=0.1 m/s CPDAT32 Tool[1]:SMC Base[0] ;%{PE}
          ;FOLD Parameters ;%{h}
          ;Params IlfProvider=kukaroboter.basistech.inlineforms.movement.spline; Kuka.IsGlobalPoint=False; Kuka.PointName=P242; Kuka.BlendingEnabled=False; Kuka.MoveDataName=CPDAT32; Kuka.VelocityPath=0.1; Kuka.VelocityFieldEnabled=True; Kuka.ColDetectFieldEnabled=True; Kuka.CurrentCDSetIndex=0; Kuka.MovementParameterFieldEnabled=True; IlfCommand=SLIN
          ;ENDFOLD
          SLIN XP242 WITH $VEL = SVEL_CP(0.1, , LCPDAT32), $TOOL = STOOL2(FP242), $BASE = SBASE(FP242.BASE_NO), $IPO_MODE = SIPO_MODE(FP242.IPO_FRAME), $LOAD = SLOAD(FP242.TOOL_NO), $ACC = SACC_CP(LCPDAT32), $ORI_TYPE = SORI_TYP(LCPDAT32), $APO = SAPO(LCPDAT32), $JERK = SJERK(LCPDAT32), $COLLMON_TOL_PRO[1] = USE_CM_PRO_VALUES(0)
          ;ENDFOLD
          ;FOLD Gripper SET [1]Gripper1 State=[2]CERRADA Wait 0.2[s] Check with Strategy 1 ;%{PE}
          ;FOLD Parameters Parameters ;%{h}
          ;Params IlfProvider=GripperTech.GripperSet;setgripper=1;setstate=2;setcont=nocont;waittime=0.2;errorstrategy=1
          ;ENDFOLD
          GRPg_SetStateAndCheck(1, 2, 0.2, 1)
          ;ENDFOLDinitialPosition
          ;FOLD SLIN P142 Vel=0.1 m/s CPDAT33 Tool[1]:SMC Base[0] ;%{PE}
          ;FOLD Parameters ;%{h}s
          ;Params IlfProvider=kukaroboter.basistech.inlineforms.movement.spline; Kuka.IsGlobalPoint=False; Kuka.PointName=P142; Kuka.BlendingEnabled=False; Kuka.MoveDataName=CPDAT33; Kuka.VelocityPath=0.1; Kuka.VelocityFieldEnabled=True; Kuka.ColDetectFieldEnabled=True; Kuka.CurrentCDSetIndex=0; Kuka.MovementParameterFieldEnabled=True; IlfCommand=SLIN
          ;ENDFOLD
          SLIN XP142 WITH $VEL = SVEL_CP(0.1, , LCPDAT33), $TOOL = STOOL2(FP142), $BASE = SBASE(FP142.BASE_NO), $IPO_MODE = SIPO_MODE(FP142.IPO_FRAME), $LOAD = SLOAD(FP142.TOOL_NO), $ACC = SACC_CP(LCPDAT33), $ORI_TYPE = SORI_TYP(LCPDAT33), $APO = SAPO(LCPDAT33), $JERK = SJERK(LCPDAT33), $COLLMON_TOL_PRO[1] = USE_CM_PRO_VALUES(0)
          ;ENDFOLD
          ;FOLD SPTP P500 Vel=100 % PDAT19 Tool[1]:SMC Base[0] ;%{PE}
          ;FOLD Parameters ;%{h}
          ;Params IlfProvider=kukaroboter.basistech.inlineforms.movement.spline; Kuka.IsGlobalPoint=False; Kuka.PointName=P500; Kuka.BlendingEnabled=False; Kuka.MoveDataPtpName=PDAT19; Kuka.VelocityPtp=100; Kuka.VelocityFieldEnabled=True; Kuka.ColDetectFieldEnabled=True; Kuka.CurrentCDSetIndex=0; Kuka.MovementParameterFieldEnabled=True; IlfCommand=SPTP
          ;ENDFOLD
          SPTP XP500 WITH $VEL_AXIS[1] = SVEL_JOINT(100.0), $TOOL = STOOL2(FP500), $BASE = SBASE(FP500.BASE_NO), $IPO_MODE = SIPO_MODE(FP500.IPO_FRAME), $LOAD = SLOAD(FP500.TOOL_NO), $ACC_AXIS[1] = SACC_JOINT(PPDAT19), $APO = SAPO_PTP(PPDAT19), $GEAR_JERK[1] = SGEAR_JERK(PPDAT19), $COLLMON_TOL_PRO[1] = USE_CM_PRO_VALUES(0)
          ;ENDFOLD
          ;FOLD Gripper SET [1]Gripper1 State=[1]ABIERTA Wait 0.2[s] Check with Strategy 1 ;%{PE}
          ;FOLD Parameters Parameters ;%{h}
          ;Params IlfProvider=GripperTech.GripperSet;setgripper=1;setstate=1;setcont=nocont;waittime=0.2;errorstrategy=1
          ;ENDFOLD
          GRPg_SetStateAndCheck(1, 1, 0.2, 1)
          ;ENDFOLD
      ENDIF
      IF eatPosition == 43 THEN
          ;FOLD SPTP P143 Vel=100 % PDAT1 Tool[1]:SMC Base[0] ;%{PE}
          ;FOLD Parameters ;%{h}
          ;Params IlfProvider=kukaroboter.basistech.inlineforms.movement.spline; Kuka.IsGlobalPoint=False; Kuka.PointName=P143; Kuka.BlendingEnabled=False; Kuka.MoveDataPtpName=PDAT1; Kuka.VelocityPtp=100; Kuka.VelocityFieldEnabled=True; Kuka.ColDetectFieldEnabled=True; Kuka.CurrentCDSetIndex=0; Kuka.MovementParameterFieldEnabled=True; IlfCommand=SPTP
          ;ENDFOLD
          SPTP XP143 WITH $VEL_AXIS[1] = SVEL_JOINT(100.0), $TOOL = STOOL2(FP143), $BASE = SBASE(FP143.BASE_NO), $IPO_MODE = SIPO_MODE(FP143.IPO_FRAME), $LOAD = SLOAD(FP143.TOOL_NO), $ACC_AXIS[1] = SACC_JOINT(PPDAT1), $APO = SAPO_PTP(PPDAT1), $GEAR_JERK[1] = SGEAR_JERK(PPDAT1), $COLLMON_TOL_PRO[1] = USE_CM_PRO_VALUES(0)
          ;ENDFOLD
          ;FOLD SLIN P243 Vel=0.1 m/s CPDAT32 Tool[1]:SMC Base[0] ;%{PE}
          ;FOLD Parameters ;%{h}
          ;Params IlfProvider=kukaroboter.basistech.inlineforms.movement.spline; Kuka.IsGlobalPoint=False; Kuka.PointName=P243; Kuka.BlendingEnabled=False; Kuka.MoveDataName=CPDAT32; Kuka.VelocityPath=0.1; Kuka.VelocityFieldEnabled=True; Kuka.ColDetectFieldEnabled=True; Kuka.CurrentCDSetIndex=0; Kuka.MovementParameterFieldEnabled=True; IlfCommand=SLIN
          ;ENDFOLD
          SLIN XP243 WITH $VEL = SVEL_CP(0.1, , LCPDAT32), $TOOL = STOOL2(FP243), $BASE = SBASE(FP243.BASE_NO), $IPO_MODE = SIPO_MODE(FP243.IPO_FRAME), $LOAD = SLOAD(FP243.TOOL_NO), $ACC = SACC_CP(LCPDAT32), $ORI_TYPE = SORI_TYP(LCPDAT32), $APO = SAPO(LCPDAT32), $JERK = SJERK(LCPDAT32), $COLLMON_TOL_PRO[1] = USE_CM_PRO_VALUES(0)
          ;ENDFOLD
          ;FOLD Gripper SET [1]Gripper1 State=[2]CERRADA Wait 0.2[s] Check with Strategy 1 ;%{PE}
          ;FOLD Parameters Parameters ;%{h}
          ;Params IlfProvider=GripperTech.GripperSet;setgripper=1;setstate=2;setcont=nocont;waittime=0.2;errorstrategy=1
          ;ENDFOLD
          GRPg_SetStateAndCheck(1, 2, 0.2, 1)
          ;ENDFOLDinitialPosition
          ;FOLD SLIN P143 Vel=0.1 m/s CPDAT33 Tool[1]:SMC Base[0] ;%{PE}
          ;FOLD Parameters ;%{h}s
          ;Params IlfProvider=kukaroboter.basistech.inlineforms.movement.spline; Kuka.IsGlobalPoint=False; Kuka.PointName=P143; Kuka.BlendingEnabled=False; Kuka.MoveDataName=CPDAT33; Kuka.VelocityPath=0.1; Kuka.VelocityFieldEnabled=True; Kuka.ColDetectFieldEnabled=True; Kuka.CurrentCDSetIndex=0; Kuka.MovementParameterFieldEnabled=True; IlfCommand=SLIN
          ;ENDFOLD
          SLIN XP143 WITH $VEL = SVEL_CP(0.1, , LCPDAT33), $TOOL = STOOL2(FP143), $BASE = SBASE(FP143.BASE_NO), $IPO_MODE = SIPO_MODE(FP143.IPO_FRAME), $LOAD = SLOAD(FP143.TOOL_NO), $ACC = SACC_CP(LCPDAT33), $ORI_TYPE = SORI_TYP(LCPDAT33), $APO = SAPO(LCPDAT33), $JERK = SJERK(LCPDAT33), $COLLMON_TOL_PRO[1] = USE_CM_PRO_VALUES(0)
          ;ENDFOLD
          ;FOLD SPTP P500 Vel=100 % PDAT19 Tool[1]:SMC Base[0] ;%{PE}
          ;FOLD Parameters ;%{h}
          ;Params IlfProvider=kukaroboter.basistech.inlineforms.movement.spline; Kuka.IsGlobalPoint=False; Kuka.PointName=P500; Kuka.BlendingEnabled=False; Kuka.MoveDataPtpName=PDAT19; Kuka.VelocityPtp=100; Kuka.VelocityFieldEnabled=True; Kuka.ColDetectFieldEnabled=True; Kuka.CurrentCDSetIndex=0; Kuka.MovementParameterFieldEnabled=True; IlfCommand=SPTP
          ;ENDFOLD
          SPTP XP500 WITH $VEL_AXIS[1] = SVEL_JOINT(100.0), $TOOL = STOOL2(FP500), $BASE = SBASE(FP500.BASE_NO), $IPO_MODE = SIPO_MODE(FP500.IPO_FRAME), $LOAD = SLOAD(FP500.TOOL_NO), $ACC_AXIS[1] = SACC_JOINT(PPDAT19), $APO = SAPO_PTP(PPDAT19), $GEAR_JERK[1] = SGEAR_JERK(PPDAT19), $COLLMON_TOL_PRO[1] = USE_CM_PRO_VALUES(0)
          ;ENDFOLD
          ;FOLD Gripper SET [1]Gripper1 State=[1]ABIERTA Wait 0.2[s] Check with Strategy 1 ;%{PE}
          ;FOLD Parameters Parameters ;%{h}
          ;Params IlfProvider=GripperTech.GripperSet;setgripper=1;setstate=1;setcont=nocont;waittime=0.2;errorstrategy=1
          ;ENDFOLD
          GRPg_SetStateAndCheck(1, 1, 0.2, 1)
          ;ENDFOLD
      ENDIF
      IF eatPosition == 44 THEN
          ;FOLD SPTP P144 Vel=100 % PDAT1 Tool[1]:SMC Base[0] ;%{PE}
          ;FOLD Parameters ;%{h}
          ;Params IlfProvider=kukaroboter.basistech.inlineforms.movement.spline; Kuka.IsGlobalPoint=False; Kuka.PointName=P144; Kuka.BlendingEnabled=False; Kuka.MoveDataPtpName=PDAT1; Kuka.VelocityPtp=100; Kuka.VelocityFieldEnabled=True; Kuka.ColDetectFieldEnabled=True; Kuka.CurrentCDSetIndex=0; Kuka.MovementParameterFieldEnabled=True; IlfCommand=SPTP
          ;ENDFOLD
          SPTP XP144 WITH $VEL_AXIS[1] = SVEL_JOINT(100.0), $TOOL = STOOL2(FP144), $BASE = SBASE(FP144.BASE_NO), $IPO_MODE = SIPO_MODE(FP144.IPO_FRAME), $LOAD = SLOAD(FP144.TOOL_NO), $ACC_AXIS[1] = SACC_JOINT(PPDAT1), $APO = SAPO_PTP(PPDAT1), $GEAR_JERK[1] = SGEAR_JERK(PPDAT1), $COLLMON_TOL_PRO[1] = USE_CM_PRO_VALUES(0)
          ;ENDFOLD
          ;FOLD SLIN P244 Vel=0.1 m/s CPDAT32 Tool[1]:SMC Base[0] ;%{PE}
          ;FOLD Parameters ;%{h}
          ;Params IlfProvider=kukaroboter.basistech.inlineforms.movement.spline; Kuka.IsGlobalPoint=False; Kuka.PointName=P244; Kuka.BlendingEnabled=False; Kuka.MoveDataName=CPDAT32; Kuka.VelocityPath=0.1; Kuka.VelocityFieldEnabled=True; Kuka.ColDetectFieldEnabled=True; Kuka.CurrentCDSetIndex=0; Kuka.MovementParameterFieldEnabled=True; IlfCommand=SLIN
          ;ENDFOLD
          SLIN XP244 WITH $VEL = SVEL_CP(0.1, , LCPDAT32), $TOOL = STOOL2(FP244), $BASE = SBASE(FP244.BASE_NO), $IPO_MODE = SIPO_MODE(FP244.IPO_FRAME), $LOAD = SLOAD(FP244.TOOL_NO), $ACC = SACC_CP(LCPDAT32), $ORI_TYPE = SORI_TYP(LCPDAT32), $APO = SAPO(LCPDAT32), $JERK = SJERK(LCPDAT32), $COLLMON_TOL_PRO[1] = USE_CM_PRO_VALUES(0)
          ;ENDFOLD
          ;FOLD Gripper SET [1]Gripper1 State=[2]CERRADA Wait 0.2[s] Check with Strategy 1 ;%{PE}
          ;FOLD Parameters Parameters ;%{h}
          ;Params IlfProvider=GripperTech.GripperSet;setgripper=1;setstate=2;setcont=nocont;waittime=0.2;errorstrategy=1
          ;ENDFOLD
          GRPg_SetStateAndCheck(1, 2, 0.2, 1)
          ;ENDFOLDinitialPosition
          ;FOLD SLIN P144 Vel=0.1 m/s CPDAT33 Tool[1]:SMC Base[0] ;%{PE}
          ;FOLD Parameters ;%{h}s
          ;Params IlfProvider=kukaroboter.basistech.inlineforms.movement.spline; Kuka.IsGlobalPoint=False; Kuka.PointName=P144; Kuka.BlendingEnabled=False; Kuka.MoveDataName=CPDAT33; Kuka.VelocityPath=0.1; Kuka.VelocityFieldEnabled=True; Kuka.ColDetectFieldEnabled=True; Kuka.CurrentCDSetIndex=0; Kuka.MovementParameterFieldEnabled=True; IlfCommand=SLIN
          ;ENDFOLD
          SLIN XP144 WITH $VEL = SVEL_CP(0.1, , LCPDAT33), $TOOL = STOOL2(FP144), $BASE = SBASE(FP144.BASE_NO), $IPO_MODE = SIPO_MODE(FP144.IPO_FRAME), $LOAD = SLOAD(FP144.TOOL_NO), $ACC = SACC_CP(LCPDAT33), $ORI_TYPE = SORI_TYP(LCPDAT33), $APO = SAPO(LCPDAT33), $JERK = SJERK(LCPDAT33), $COLLMON_TOL_PRO[1] = USE_CM_PRO_VALUES(0)
          ;ENDFOLD
          ;FOLD SPTP P500 Vel=100 % PDAT19 Tool[1]:SMC Base[0] ;%{PE}
          ;FOLD Parameters ;%{h}
          ;Params IlfProvider=kukaroboter.basistech.inlineforms.movement.spline; Kuka.IsGlobalPoint=False; Kuka.PointName=P500; Kuka.BlendingEnabled=False; Kuka.MoveDataPtpName=PDAT19; Kuka.VelocityPtp=100; Kuka.VelocityFieldEnabled=True; Kuka.ColDetectFieldEnabled=True; Kuka.CurrentCDSetIndex=0; Kuka.MovementParameterFieldEnabled=True; IlfCommand=SPTP
          ;ENDFOLD
          SPTP XP500 WITH $VEL_AXIS[1] = SVEL_JOINT(100.0), $TOOL = STOOL2(FP500), $BASE = SBASE(FP500.BASE_NO), $IPO_MODE = SIPO_MODE(FP500.IPO_FRAME), $LOAD = SLOAD(FP500.TOOL_NO), $ACC_AXIS[1] = SACC_JOINT(PPDAT19), $APO = SAPO_PTP(PPDAT19), $GEAR_JERK[1] = SGEAR_JERK(PPDAT19), $COLLMON_TOL_PRO[1] = USE_CM_PRO_VALUES(0)
          ;ENDFOLD
          ;FOLD Gripper SET [1]Gripper1 State=[1]ABIERTA Wait 0.2[s] Check with Strategy 1 ;%{PE}
          ;FOLD Parameters Parameters ;%{h}
          ;Params IlfProvider=GripperTech.GripperSet;setgripper=1;setstate=1;setcont=nocont;waittime=0.2;errorstrategy=1
          ;ENDFOLD
          GRPg_SetStateAndCheck(1, 1, 0.2, 1)
          ;ENDFOLD
      ENDIF
      IF eatPosition == 45 THEN
          ;FOLD SPTP P145 Vel=100 % PDAT1 Tool[1]:SMC Base[0] ;%{PE}
          ;FOLD Parameters ;%{h}
          ;Params IlfProvider=kukaroboter.basistech.inlineforms.movement.spline; Kuka.IsGlobalPoint=False; Kuka.PointName=P145; Kuka.BlendingEnabled=False; Kuka.MoveDataPtpName=PDAT1; Kuka.VelocityPtp=100; Kuka.VelocityFieldEnabled=True; Kuka.ColDetectFieldEnabled=True; Kuka.CurrentCDSetIndex=0; Kuka.MovementParameterFieldEnabled=True; IlfCommand=SPTP
          ;ENDFOLD
          SPTP XP145 WITH $VEL_AXIS[1] = SVEL_JOINT(100.0), $TOOL = STOOL2(FP145), $BASE = SBASE(FP145.BASE_NO), $IPO_MODE = SIPO_MODE(FP145.IPO_FRAME), $LOAD = SLOAD(FP145.TOOL_NO), $ACC_AXIS[1] = SACC_JOINT(PPDAT1), $APO = SAPO_PTP(PPDAT1), $GEAR_JERK[1] = SGEAR_JERK(PPDAT1), $COLLMON_TOL_PRO[1] = USE_CM_PRO_VALUES(0)
          ;ENDFOLD
          ;FOLD SLIN P245 Vel=0.1 m/s CPDAT32 Tool[1]:SMC Base[0] ;%{PE}
          ;FOLD Parameters ;%{h}
          ;Params IlfProvider=kukaroboter.basistech.inlineforms.movement.spline; Kuka.IsGlobalPoint=False; Kuka.PointName=P245; Kuka.BlendingEnabled=False; Kuka.MoveDataName=CPDAT32; Kuka.VelocityPath=0.1; Kuka.VelocityFieldEnabled=True; Kuka.ColDetectFieldEnabled=True; Kuka.CurrentCDSetIndex=0; Kuka.MovementParameterFieldEnabled=True; IlfCommand=SLIN
          ;ENDFOLD
          SLIN XP245 WITH $VEL = SVEL_CP(0.1, , LCPDAT32), $TOOL = STOOL2(FP245), $BASE = SBASE(FP245.BASE_NO), $IPO_MODE = SIPO_MODE(FP245.IPO_FRAME), $LOAD = SLOAD(FP245.TOOL_NO), $ACC = SACC_CP(LCPDAT32), $ORI_TYPE = SORI_TYP(LCPDAT32), $APO = SAPO(LCPDAT32), $JERK = SJERK(LCPDAT32), $COLLMON_TOL_PRO[1] = USE_CM_PRO_VALUES(0)
          ;ENDFOLD
          ;FOLD Gripper SET [1]Gripper1 State=[2]CERRADA Wait 0.2[s] Check with Strategy 1 ;%{PE}
          ;FOLD Parameters Parameters ;%{h}
          ;Params IlfProvider=GripperTech.GripperSet;setgripper=1;setstate=2;setcont=nocont;waittime=0.2;errorstrategy=1
          ;ENDFOLD
          GRPg_SetStateAndCheck(1, 2, 0.2, 1)
          ;ENDFOLDinitialPosition
          ;FOLD SLIN P145 Vel=0.1 m/s CPDAT33 Tool[1]:SMC Base[0] ;%{PE}
          ;FOLD Parameters ;%{h}s
          ;Params IlfProvider=kukaroboter.basistech.inlineforms.movement.spline; Kuka.IsGlobalPoint=False; Kuka.PointName=P145; Kuka.BlendingEnabled=False; Kuka.MoveDataName=CPDAT33; Kuka.VelocityPath=0.1; Kuka.VelocityFieldEnabled=True; Kuka.ColDetectFieldEnabled=True; Kuka.CurrentCDSetIndex=0; Kuka.MovementParameterFieldEnabled=True; IlfCommand=SLIN
          ;ENDFOLD
          SLIN XP145 WITH $VEL = SVEL_CP(0.1, , LCPDAT33), $TOOL = STOOL2(FP145), $BASE = SBASE(FP145.BASE_NO), $IPO_MODE = SIPO_MODE(FP145.IPO_FRAME), $LOAD = SLOAD(FP145.TOOL_NO), $ACC = SACC_CP(LCPDAT33), $ORI_TYPE = SORI_TYP(LCPDAT33), $APO = SAPO(LCPDAT33), $JERK = SJERK(LCPDAT33), $COLLMON_TOL_PRO[1] = USE_CM_PRO_VALUES(0)
          ;ENDFOLD
          ;FOLD SPTP P500 Vel=100 % PDAT19 Tool[1]:SMC Base[0] ;%{PE}
          ;FOLD Parameters ;%{h}
          ;Params IlfProvider=kukaroboter.basistech.inlineforms.movement.spline; Kuka.IsGlobalPoint=False; Kuka.PointName=P500; Kuka.BlendingEnabled=False; Kuka.MoveDataPtpName=PDAT19; Kuka.VelocityPtp=100; Kuka.VelocityFieldEnabled=True; Kuka.ColDetectFieldEnabled=True; Kuka.CurrentCDSetIndex=0; Kuka.MovementParameterFieldEnabled=True; IlfCommand=SPTP
          ;ENDFOLD
          SPTP XP500 WITH $VEL_AXIS[1] = SVEL_JOINT(100.0), $TOOL = STOOL2(FP500), $BASE = SBASE(FP500.BASE_NO), $IPO_MODE = SIPO_MODE(FP500.IPO_FRAME), $LOAD = SLOAD(FP500.TOOL_NO), $ACC_AXIS[1] = SACC_JOINT(PPDAT19), $APO = SAPO_PTP(PPDAT19), $GEAR_JERK[1] = SGEAR_JERK(PPDAT19), $COLLMON_TOL_PRO[1] = USE_CM_PRO_VALUES(0)
          ;ENDFOLD
          ;FOLD Gripper SET [1]Gripper1 State=[1]ABIERTA Wait 0.2[s] Check with Strategy 1 ;%{PE}
          ;FOLD Parameters Parameters ;%{h}
          ;Params IlfProvider=GripperTech.GripperSet;setgripper=1;setstate=1;setcont=nocont;waittime=0.2;errorstrategy=1
          ;ENDFOLD
          GRPg_SetStateAndCheck(1, 1, 0.2, 1)
          ;ENDFOLD
      ENDIF
      IF eatPosition == 46 THEN
          ;FOLD SPTP P146 Vel=100 % PDAT1 Tool[1]:SMC Base[0] ;%{PE}
          ;FOLD Parameters ;%{h}
          ;Params IlfProvider=kukaroboter.basistech.inlineforms.movement.spline; Kuka.IsGlobalPoint=False; Kuka.PointName=P146; Kuka.BlendingEnabled=False; Kuka.MoveDataPtpName=PDAT1; Kuka.VelocityPtp=100; Kuka.VelocityFieldEnabled=True; Kuka.ColDetectFieldEnabled=True; Kuka.CurrentCDSetIndex=0; Kuka.MovementParameterFieldEnabled=True; IlfCommand=SPTP
          ;ENDFOLD
          SPTP XP146 WITH $VEL_AXIS[1] = SVEL_JOINT(100.0), $TOOL = STOOL2(FP146), $BASE = SBASE(FP146.BASE_NO), $IPO_MODE = SIPO_MODE(FP146.IPO_FRAME), $LOAD = SLOAD(FP146.TOOL_NO), $ACC_AXIS[1] = SACC_JOINT(PPDAT1), $APO = SAPO_PTP(PPDAT1), $GEAR_JERK[1] = SGEAR_JERK(PPDAT1), $COLLMON_TOL_PRO[1] = USE_CM_PRO_VALUES(0)
          ;ENDFOLD
          ;FOLD SLIN P246 Vel=0.1 m/s CPDAT32 Tool[1]:SMC Base[0] ;%{PE}
          ;FOLD Parameters ;%{h}
          ;Params IlfProvider=kukaroboter.basistech.inlineforms.movement.spline; Kuka.IsGlobalPoint=False; Kuka.PointName=P246; Kuka.BlendingEnabled=False; Kuka.MoveDataName=CPDAT32; Kuka.VelocityPath=0.1; Kuka.VelocityFieldEnabled=True; Kuka.ColDetectFieldEnabled=True; Kuka.CurrentCDSetIndex=0; Kuka.MovementParameterFieldEnabled=True; IlfCommand=SLIN
          ;ENDFOLD
          SLIN XP246 WITH $VEL = SVEL_CP(0.1, , LCPDAT32), $TOOL = STOOL2(FP246), $BASE = SBASE(FP246.BASE_NO), $IPO_MODE = SIPO_MODE(FP246.IPO_FRAME), $LOAD = SLOAD(FP246.TOOL_NO), $ACC = SACC_CP(LCPDAT32), $ORI_TYPE = SORI_TYP(LCPDAT32), $APO = SAPO(LCPDAT32), $JERK = SJERK(LCPDAT32), $COLLMON_TOL_PRO[1] = USE_CM_PRO_VALUES(0)
          ;ENDFOLD
          ;FOLD Gripper SET [1]Gripper1 State=[2]CERRADA Wait 0.2[s] Check with Strategy 1 ;%{PE}
          ;FOLD Parameters Parameters ;%{h}
          ;Params IlfProvider=GripperTech.GripperSet;setgripper=1;setstate=2;setcont=nocont;waittime=0.2;errorstrategy=1
          ;ENDFOLD
          GRPg_SetStateAndCheck(1, 2, 0.2, 1)
          ;ENDFOLDinitialPosition
          ;FOLD SLIN P146 Vel=0.1 m/s CPDAT33 Tool[1]:SMC Base[0] ;%{PE}
          ;FOLD Parameters ;%{h}s
          ;Params IlfProvider=kukaroboter.basistech.inlineforms.movement.spline; Kuka.IsGlobalPoint=False; Kuka.PointName=P146; Kuka.BlendingEnabled=False; Kuka.MoveDataName=CPDAT33; Kuka.VelocityPath=0.1; Kuka.VelocityFieldEnabled=True; Kuka.ColDetectFieldEnabled=True; Kuka.CurrentCDSetIndex=0; Kuka.MovementParameterFieldEnabled=True; IlfCommand=SLIN
          ;ENDFOLD
          SLIN XP146 WITH $VEL = SVEL_CP(0.1, , LCPDAT33), $TOOL = STOOL2(FP146), $BASE = SBASE(FP146.BASE_NO), $IPO_MODE = SIPO_MODE(FP146.IPO_FRAME), $LOAD = SLOAD(FP146.TOOL_NO), $ACC = SACC_CP(LCPDAT33), $ORI_TYPE = SORI_TYP(LCPDAT33), $APO = SAPO(LCPDAT33), $JERK = SJERK(LCPDAT33), $COLLMON_TOL_PRO[1] = USE_CM_PRO_VALUES(0)
          ;ENDFOLD
          ;FOLD SPTP P500 Vel=100 % PDAT19 Tool[1]:SMC Base[0] ;%{PE}
          ;FOLD Parameters ;%{h}
          ;Params IlfProvider=kukaroboter.basistech.inlineforms.movement.spline; Kuka.IsGlobalPoint=False; Kuka.PointName=P500; Kuka.BlendingEnabled=False; Kuka.MoveDataPtpName=PDAT19; Kuka.VelocityPtp=100; Kuka.VelocityFieldEnabled=True; Kuka.ColDetectFieldEnabled=True; Kuka.CurrentCDSetIndex=0; Kuka.MovementParameterFieldEnabled=True; IlfCommand=SPTP
          ;ENDFOLD
          SPTP XP500 WITH $VEL_AXIS[1] = SVEL_JOINT(100.0), $TOOL = STOOL2(FP500), $BASE = SBASE(FP500.BASE_NO), $IPO_MODE = SIPO_MODE(FP500.IPO_FRAME), $LOAD = SLOAD(FP500.TOOL_NO), $ACC_AXIS[1] = SACC_JOINT(PPDAT19), $APO = SAPO_PTP(PPDAT19), $GEAR_JERK[1] = SGEAR_JERK(PPDAT19), $COLLMON_TOL_PRO[1] = USE_CM_PRO_VALUES(0)
          ;ENDFOLD
          ;FOLD Gripper SET [1]Gripper1 State=[1]ABIERTA Wait 0.2[s] Check with Strategy 1 ;%{PE}
          ;FOLD Parameters Parameters ;%{h}
          ;Params IlfProvider=GripperTech.GripperSet;setgripper=1;setstate=1;setcont=nocont;waittime=0.2;errorstrategy=1
          ;ENDFOLD
          GRPg_SetStateAndCheck(1, 1, 0.2, 1)
          ;ENDFOLD
      ENDIF
      IF eatPosition == 47 THEN
          ;FOLD SPTP P147 Vel=100 % PDAT1 Tool[1]:SMC Base[0] ;%{PE}
          ;FOLD Parameters ;%{h}
          ;Params IlfProvider=kukaroboter.basistech.inlineforms.movement.spline; Kuka.IsGlobalPoint=False; Kuka.PointName=P147; Kuka.BlendingEnabled=False; Kuka.MoveDataPtpName=PDAT1; Kuka.VelocityPtp=100; Kuka.VelocityFieldEnabled=True; Kuka.ColDetectFieldEnabled=True; Kuka.CurrentCDSetIndex=0; Kuka.MovementParameterFieldEnabled=True; IlfCommand=SPTP
          ;ENDFOLD
          SPTP XP147 WITH $VEL_AXIS[1] = SVEL_JOINT(100.0), $TOOL = STOOL2(FP147), $BASE = SBASE(FP147.BASE_NO), $IPO_MODE = SIPO_MODE(FP147.IPO_FRAME), $LOAD = SLOAD(FP147.TOOL_NO), $ACC_AXIS[1] = SACC_JOINT(PPDAT1), $APO = SAPO_PTP(PPDAT1), $GEAR_JERK[1] = SGEAR_JERK(PPDAT1), $COLLMON_TOL_PRO[1] = USE_CM_PRO_VALUES(0)
          ;ENDFOLD
          ;FOLD SLIN P247 Vel=0.1 m/s CPDAT32 Tool[1]:SMC Base[0] ;%{PE}
          ;FOLD Parameters ;%{h}
          ;Params IlfProvider=kukaroboter.basistech.inlineforms.movement.spline; Kuka.IsGlobalPoint=False; Kuka.PointName=P247; Kuka.BlendingEnabled=False; Kuka.MoveDataName=CPDAT32; Kuka.VelocityPath=0.1; Kuka.VelocityFieldEnabled=True; Kuka.ColDetectFieldEnabled=True; Kuka.CurrentCDSetIndex=0; Kuka.MovementParameterFieldEnabled=True; IlfCommand=SLIN
          ;ENDFOLD
          SLIN XP247 WITH $VEL = SVEL_CP(0.1, , LCPDAT32), $TOOL = STOOL2(FP247), $BASE = SBASE(FP247.BASE_NO), $IPO_MODE = SIPO_MODE(FP247.IPO_FRAME), $LOAD = SLOAD(FP247.TOOL_NO), $ACC = SACC_CP(LCPDAT32), $ORI_TYPE = SORI_TYP(LCPDAT32), $APO = SAPO(LCPDAT32), $JERK = SJERK(LCPDAT32), $COLLMON_TOL_PRO[1] = USE_CM_PRO_VALUES(0)
          ;ENDFOLD
          ;FOLD Gripper SET [1]Gripper1 State=[2]CERRADA Wait 0.2[s] Check with Strategy 1 ;%{PE}
          ;FOLD Parameters Parameters ;%{h}
          ;Params IlfProvider=GripperTech.GripperSet;setgripper=1;setstate=2;setcont=nocont;waittime=0.2;errorstrategy=1
          ;ENDFOLD
          GRPg_SetStateAndCheck(1, 2, 0.2, 1)
          ;ENDFOLDinitialPosition
          ;FOLD SLIN P147 Vel=0.1 m/s CPDAT33 Tool[1]:SMC Base[0] ;%{PE}
          ;FOLD Parameters ;%{h}s
          ;Params IlfProvider=kukaroboter.basistech.inlineforms.movement.spline; Kuka.IsGlobalPoint=False; Kuka.PointName=P147; Kuka.BlendingEnabled=False; Kuka.MoveDataName=CPDAT33; Kuka.VelocityPath=0.1; Kuka.VelocityFieldEnabled=True; Kuka.ColDetectFieldEnabled=True; Kuka.CurrentCDSetIndex=0; Kuka.MovementParameterFieldEnabled=True; IlfCommand=SLIN
          ;ENDFOLD
          SLIN XP147 WITH $VEL = SVEL_CP(0.1, , LCPDAT33), $TOOL = STOOL2(FP147), $BASE = SBASE(FP147.BASE_NO), $IPO_MODE = SIPO_MODE(FP147.IPO_FRAME), $LOAD = SLOAD(FP147.TOOL_NO), $ACC = SACC_CP(LCPDAT33), $ORI_TYPE = SORI_TYP(LCPDAT33), $APO = SAPO(LCPDAT33), $JERK = SJERK(LCPDAT33), $COLLMON_TOL_PRO[1] = USE_CM_PRO_VALUES(0)
          ;ENDFOLD
          ;FOLD SPTP P500 Vel=100 % PDAT19 Tool[1]:SMC Base[0] ;%{PE}
          ;FOLD Parameters ;%{h}
          ;Params IlfProvider=kukaroboter.basistech.inlineforms.movement.spline; Kuka.IsGlobalPoint=False; Kuka.PointName=P500; Kuka.BlendingEnabled=False; Kuka.MoveDataPtpName=PDAT19; Kuka.VelocityPtp=100; Kuka.VelocityFieldEnabled=True; Kuka.ColDetectFieldEnabled=True; Kuka.CurrentCDSetIndex=0; Kuka.MovementParameterFieldEnabled=True; IlfCommand=SPTP
          ;ENDFOLD
          SPTP XP500 WITH $VEL_AXIS[1] = SVEL_JOINT(100.0), $TOOL = STOOL2(FP500), $BASE = SBASE(FP500.BASE_NO), $IPO_MODE = SIPO_MODE(FP500.IPO_FRAME), $LOAD = SLOAD(FP500.TOOL_NO), $ACC_AXIS[1] = SACC_JOINT(PPDAT19), $APO = SAPO_PTP(PPDAT19), $GEAR_JERK[1] = SGEAR_JERK(PPDAT19), $COLLMON_TOL_PRO[1] = USE_CM_PRO_VALUES(0)
          ;ENDFOLD
          ;FOLD Gripper SET [1]Gripper1 State=[1]ABIERTA Wait 0.2[s] Check with Strategy 1 ;%{PE}
          ;FOLD Parameters Parameters ;%{h}
          ;Params IlfProvider=GripperTech.GripperSet;setgripper=1;setstate=1;setcont=nocont;waittime=0.2;errorstrategy=1
          ;ENDFOLD
          GRPg_SetStateAndCheck(1, 1, 0.2, 1)
          ;ENDFOLD
      ENDIF
      IF eatPosition == 48 THEN
          ;FOLD SPTP P148 Vel=100 % PDAT1 Tool[1]:SMC Base[0] ;%{PE}
          ;FOLD Parameters ;%{h}
          ;Params IlfProvider=kukaroboter.basistech.inlineforms.movement.spline; Kuka.IsGlobalPoint=False; Kuka.PointName=P148; Kuka.BlendingEnabled=False; Kuka.MoveDataPtpName=PDAT1; Kuka.VelocityPtp=100; Kuka.VelocityFieldEnabled=True; Kuka.ColDetectFieldEnabled=True; Kuka.CurrentCDSetIndex=0; Kuka.MovementParameterFieldEnabled=True; IlfCommand=SPTP
          ;ENDFOLD
          SPTP XP148 WITH $VEL_AXIS[1] = SVEL_JOINT(100.0), $TOOL = STOOL2(FP148), $BASE = SBASE(FP148.BASE_NO), $IPO_MODE = SIPO_MODE(FP148.IPO_FRAME), $LOAD = SLOAD(FP148.TOOL_NO), $ACC_AXIS[1] = SACC_JOINT(PPDAT1), $APO = SAPO_PTP(PPDAT1), $GEAR_JERK[1] = SGEAR_JERK(PPDAT1), $COLLMON_TOL_PRO[1] = USE_CM_PRO_VALUES(0)
          ;ENDFOLD
          ;FOLD SLIN P248 Vel=0.1 m/s CPDAT32 Tool[1]:SMC Base[0] ;%{PE}
          ;FOLD Parameters ;%{h}
          ;Params IlfProvider=kukaroboter.basistech.inlineforms.movement.spline; Kuka.IsGlobalPoint=False; Kuka.PointName=P248; Kuka.BlendingEnabled=False; Kuka.MoveDataName=CPDAT32; Kuka.VelocityPath=0.1; Kuka.VelocityFieldEnabled=True; Kuka.ColDetectFieldEnabled=True; Kuka.CurrentCDSetIndex=0; Kuka.MovementParameterFieldEnabled=True; IlfCommand=SLIN
          ;ENDFOLD
          SLIN XP248 WITH $VEL = SVEL_CP(0.1, , LCPDAT32), $TOOL = STOOL2(FP248), $BASE = SBASE(FP248.BASE_NO), $IPO_MODE = SIPO_MODE(FP248.IPO_FRAME), $LOAD = SLOAD(FP248.TOOL_NO), $ACC = SACC_CP(LCPDAT32), $ORI_TYPE = SORI_TYP(LCPDAT32), $APO = SAPO(LCPDAT32), $JERK = SJERK(LCPDAT32), $COLLMON_TOL_PRO[1] = USE_CM_PRO_VALUES(0)
          ;ENDFOLD
          ;FOLD Gripper SET [1]Gripper1 State=[2]CERRADA Wait 0.2[s] Check with Strategy 1 ;%{PE}
          ;FOLD Parameters Parameters ;%{h}
          ;Params IlfProvider=GripperTech.GripperSet;setgripper=1;setstate=2;setcont=nocont;waittime=0.2;errorstrategy=1
          ;ENDFOLD
          GRPg_SetStateAndCheck(1, 2, 0.2, 1)
          ;ENDFOLDinitialPosition
          ;FOLD SLIN P148 Vel=0.1 m/s CPDAT33 Tool[1]:SMC Base[0] ;%{PE}
          ;FOLD Parameters ;%{h}s
          ;Params IlfProvider=kukaroboter.basistech.inlineforms.movement.spline; Kuka.IsGlobalPoint=False; Kuka.PointName=P148; Kuka.BlendingEnabled=False; Kuka.MoveDataName=CPDAT33; Kuka.VelocityPath=0.1; Kuka.VelocityFieldEnabled=True; Kuka.ColDetectFieldEnabled=True; Kuka.CurrentCDSetIndex=0; Kuka.MovementParameterFieldEnabled=True; IlfCommand=SLIN
          ;ENDFOLD
          SLIN XP148 WITH $VEL = SVEL_CP(0.1, , LCPDAT33), $TOOL = STOOL2(FP148), $BASE = SBASE(FP148.BASE_NO), $IPO_MODE = SIPO_MODE(FP148.IPO_FRAME), $LOAD = SLOAD(FP148.TOOL_NO), $ACC = SACC_CP(LCPDAT33), $ORI_TYPE = SORI_TYP(LCPDAT33), $APO = SAPO(LCPDAT33), $JERK = SJERK(LCPDAT33), $COLLMON_TOL_PRO[1] = USE_CM_PRO_VALUES(0)
          ;ENDFOLD
          ;FOLD SPTP P500 Vel=100 % PDAT19 Tool[1]:SMC Base[0] ;%{PE}
          ;FOLD Parameters ;%{h}
          ;Params IlfProvider=kukaroboter.basistech.inlineforms.movement.spline; Kuka.IsGlobalPoint=False; Kuka.PointName=P500; Kuka.BlendingEnabled=False; Kuka.MoveDataPtpName=PDAT19; Kuka.VelocityPtp=100; Kuka.VelocityFieldEnabled=True; Kuka.ColDetectFieldEnabled=True; Kuka.CurrentCDSetIndex=0; Kuka.MovementParameterFieldEnabled=True; IlfCommand=SPTP
          ;ENDFOLD
          SPTP XP500 WITH $VEL_AXIS[1] = SVEL_JOINT(100.0), $TOOL = STOOL2(FP500), $BASE = SBASE(FP500.BASE_NO), $IPO_MODE = SIPO_MODE(FP500.IPO_FRAME), $LOAD = SLOAD(FP500.TOOL_NO), $ACC_AXIS[1] = SACC_JOINT(PPDAT19), $APO = SAPO_PTP(PPDAT19), $GEAR_JERK[1] = SGEAR_JERK(PPDAT19), $COLLMON_TOL_PRO[1] = USE_CM_PRO_VALUES(0)
          ;ENDFOLD
          ;FOLD Gripper SET [1]Gripper1 State=[1]ABIERTA Wait 0.2[s] Check with Strategy 1 ;%{PE}
          ;FOLD Parameters Parameters ;%{h}
          ;Params IlfProvider=GripperTech.GripperSet;setgripper=1;setstate=1;setcont=nocont;waittime=0.2;errorstrategy=1
          ;ENDFOLD
          GRPg_SetStateAndCheck(1, 1, 0.2, 1)
          ;ENDFOLD
      ENDIF
      IF eatPosition == 49 THEN
          ;FOLD SPTP P149 Vel=100 % PDAT1 Tool[1]:SMC Base[0] ;%{PE}
          ;FOLD Parameters ;%{h}
          ;Params IlfProvider=kukaroboter.basistech.inlineforms.movement.spline; Kuka.IsGlobalPoint=False; Kuka.PointName=P149; Kuka.BlendingEnabled=False; Kuka.MoveDataPtpName=PDAT1; Kuka.VelocityPtp=100; Kuka.VelocityFieldEnabled=True; Kuka.ColDetectFieldEnabled=True; Kuka.CurrentCDSetIndex=0; Kuka.MovementParameterFieldEnabled=True; IlfCommand=SPTP
          ;ENDFOLD
          SPTP XP149 WITH $VEL_AXIS[1] = SVEL_JOINT(100.0), $TOOL = STOOL2(FP149), $BASE = SBASE(FP149.BASE_NO), $IPO_MODE = SIPO_MODE(FP149.IPO_FRAME), $LOAD = SLOAD(FP149.TOOL_NO), $ACC_AXIS[1] = SACC_JOINT(PPDAT1), $APO = SAPO_PTP(PPDAT1), $GEAR_JERK[1] = SGEAR_JERK(PPDAT1), $COLLMON_TOL_PRO[1] = USE_CM_PRO_VALUES(0)
          ;ENDFOLD
          ;FOLD SLIN P249 Vel=0.1 m/s CPDAT32 Tool[1]:SMC Base[0] ;%{PE}
          ;FOLD Parameters ;%{h}
          ;Params IlfProvider=kukaroboter.basistech.inlineforms.movement.spline; Kuka.IsGlobalPoint=False; Kuka.PointName=P249; Kuka.BlendingEnabled=False; Kuka.MoveDataName=CPDAT32; Kuka.VelocityPath=0.1; Kuka.VelocityFieldEnabled=True; Kuka.ColDetectFieldEnabled=True; Kuka.CurrentCDSetIndex=0; Kuka.MovementParameterFieldEnabled=True; IlfCommand=SLIN
          ;ENDFOLD
          SLIN XP249 WITH $VEL = SVEL_CP(0.1, , LCPDAT32), $TOOL = STOOL2(FP249), $BASE = SBASE(FP249.BASE_NO), $IPO_MODE = SIPO_MODE(FP249.IPO_FRAME), $LOAD = SLOAD(FP249.TOOL_NO), $ACC = SACC_CP(LCPDAT32), $ORI_TYPE = SORI_TYP(LCPDAT32), $APO = SAPO(LCPDAT32), $JERK = SJERK(LCPDAT32), $COLLMON_TOL_PRO[1] = USE_CM_PRO_VALUES(0)
          ;ENDFOLD
          ;FOLD Gripper SET [1]Gripper1 State=[2]CERRADA Wait 0.2[s] Check with Strategy 1 ;%{PE}
          ;FOLD Parameters Parameters ;%{h}
          ;Params IlfProvider=GripperTech.GripperSet;setgripper=1;setstate=2;setcont=nocont;waittime=0.2;errorstrategy=1
          ;ENDFOLD
          GRPg_SetStateAndCheck(1, 2, 0.2, 1)
          ;ENDFOLDinitialPosition
          ;FOLD SLIN P149 Vel=0.1 m/s CPDAT33 Tool[1]:SMC Base[0] ;%{PE}
          ;FOLD Parameters ;%{h}s
          ;Params IlfProvider=kukaroboter.basistech.inlineforms.movement.spline; Kuka.IsGlobalPoint=False; Kuka.PointName=P149; Kuka.BlendingEnabled=False; Kuka.MoveDataName=CPDAT33; Kuka.VelocityPath=0.1; Kuka.VelocityFieldEnabled=True; Kuka.ColDetectFieldEnabled=True; Kuka.CurrentCDSetIndex=0; Kuka.MovementParameterFieldEnabled=True; IlfCommand=SLIN
          ;ENDFOLD
          SLIN XP149 WITH $VEL = SVEL_CP(0.1, , LCPDAT33), $TOOL = STOOL2(FP149), $BASE = SBASE(FP149.BASE_NO), $IPO_MODE = SIPO_MODE(FP149.IPO_FRAME), $LOAD = SLOAD(FP149.TOOL_NO), $ACC = SACC_CP(LCPDAT33), $ORI_TYPE = SORI_TYP(LCPDAT33), $APO = SAPO(LCPDAT33), $JERK = SJERK(LCPDAT33), $COLLMON_TOL_PRO[1] = USE_CM_PRO_VALUES(0)
          ;ENDFOLD
          ;FOLD SPTP P500 Vel=100 % PDAT19 Tool[1]:SMC Base[0] ;%{PE}
          ;FOLD Parameters ;%{h}
          ;Params IlfProvider=kukaroboter.basistech.inlineforms.movement.spline; Kuka.IsGlobalPoint=False; Kuka.PointName=P500; Kuka.BlendingEnabled=False; Kuka.MoveDataPtpName=PDAT19; Kuka.VelocityPtp=100; Kuka.VelocityFieldEnabled=True; Kuka.ColDetectFieldEnabled=True; Kuka.CurrentCDSetIndex=0; Kuka.MovementParameterFieldEnabled=True; IlfCommand=SPTP
          ;ENDFOLD
          SPTP XP500 WITH $VEL_AXIS[1] = SVEL_JOINT(100.0), $TOOL = STOOL2(FP500), $BASE = SBASE(FP500.BASE_NO), $IPO_MODE = SIPO_MODE(FP500.IPO_FRAME), $LOAD = SLOAD(FP500.TOOL_NO), $ACC_AXIS[1] = SACC_JOINT(PPDAT19), $APO = SAPO_PTP(PPDAT19), $GEAR_JERK[1] = SGEAR_JERK(PPDAT19), $COLLMON_TOL_PRO[1] = USE_CM_PRO_VALUES(0)
          ;ENDFOLD
          ;FOLD Gripper SET [1]Gripper1 State=[1]ABIERTA Wait 0.2[s] Check with Strategy 1 ;%{PE}
          ;FOLD Parameters Parameters ;%{h}
          ;Params IlfProvider=GripperTech.GripperSet;setgripper=1;setstate=1;setcont=nocont;waittime=0.2;errorstrategy=1
          ;ENDFOLD
          GRPg_SetStateAndCheck(1, 1, 0.2, 1)
          ;ENDFOLD
      ENDIF
      IF eatPosition == 50 THEN
          ;FOLD SPTP P150 Vel=100 % PDAT1 Tool[1]:SMC Base[0] ;%{PE}
          ;FOLD Parameters ;%{h}
          ;Params IlfProvider=kukaroboter.basistech.inlineforms.movement.spline; Kuka.IsGlobalPoint=False; Kuka.PointName=P150; Kuka.BlendingEnabled=False; Kuka.MoveDataPtpName=PDAT1; Kuka.VelocityPtp=100; Kuka.VelocityFieldEnabled=True; Kuka.ColDetectFieldEnabled=True; Kuka.CurrentCDSetIndex=0; Kuka.MovementParameterFieldEnabled=True; IlfCommand=SPTP
          ;ENDFOLD
          SPTP XP150 WITH $VEL_AXIS[1] = SVEL_JOINT(100.0), $TOOL = STOOL2(FP150), $BASE = SBASE(FP150.BASE_NO), $IPO_MODE = SIPO_MODE(FP150.IPO_FRAME), $LOAD = SLOAD(FP150.TOOL_NO), $ACC_AXIS[1] = SACC_JOINT(PPDAT1), $APO = SAPO_PTP(PPDAT1), $GEAR_JERK[1] = SGEAR_JERK(PPDAT1), $COLLMON_TOL_PRO[1] = USE_CM_PRO_VALUES(0)
          ;ENDFOLD
          ;FOLD SLIN P250 Vel=0.1 m/s CPDAT32 Tool[1]:SMC Base[0] ;%{PE}
          ;FOLD Parameters ;%{h}
          ;Params IlfProvider=kukaroboter.basistech.inlineforms.movement.spline; Kuka.IsGlobalPoint=False; Kuka.PointName=P250; Kuka.BlendingEnabled=False; Kuka.MoveDataName=CPDAT32; Kuka.VelocityPath=0.1; Kuka.VelocityFieldEnabled=True; Kuka.ColDetectFieldEnabled=True; Kuka.CurrentCDSetIndex=0; Kuka.MovementParameterFieldEnabled=True; IlfCommand=SLIN
          ;ENDFOLD
          SLIN XP250 WITH $VEL = SVEL_CP(0.1, , LCPDAT32), $TOOL = STOOL2(FP250), $BASE = SBASE(FP250.BASE_NO), $IPO_MODE = SIPO_MODE(FP250.IPO_FRAME), $LOAD = SLOAD(FP250.TOOL_NO), $ACC = SACC_CP(LCPDAT32), $ORI_TYPE = SORI_TYP(LCPDAT32), $APO = SAPO(LCPDAT32), $JERK = SJERK(LCPDAT32), $COLLMON_TOL_PRO[1] = USE_CM_PRO_VALUES(0)
          ;ENDFOLD
          ;FOLD Gripper SET [1]Gripper1 State=[2]CERRADA Wait 0.2[s] Check with Strategy 1 ;%{PE}
          ;FOLD Parameters Parameters ;%{h}
          ;Params IlfProvider=GripperTech.GripperSet;setgripper=1;setstate=2;setcont=nocont;waittime=0.2;errorstrategy=1
          ;ENDFOLD
          GRPg_SetStateAndCheck(1, 2, 0.2, 1)
          ;ENDFOLDinitialPosition
          ;FOLD SLIN P150 Vel=0.1 m/s CPDAT33 Tool[1]:SMC Base[0] ;%{PE}
          ;FOLD Parameters ;%{h}s
          ;Params IlfProvider=kukaroboter.basistech.inlineforms.movement.spline; Kuka.IsGlobalPoint=False; Kuka.PointName=P150; Kuka.BlendingEnabled=False; Kuka.MoveDataName=CPDAT33; Kuka.VelocityPath=0.1; Kuka.VelocityFieldEnabled=True; Kuka.ColDetectFieldEnabled=True; Kuka.CurrentCDSetIndex=0; Kuka.MovementParameterFieldEnabled=True; IlfCommand=SLIN
          ;ENDFOLD
          SLIN XP150 WITH $VEL = SVEL_CP(0.1, , LCPDAT33), $TOOL = STOOL2(FP150), $BASE = SBASE(FP150.BASE_NO), $IPO_MODE = SIPO_MODE(FP150.IPO_FRAME), $LOAD = SLOAD(FP150.TOOL_NO), $ACC = SACC_CP(LCPDAT33), $ORI_TYPE = SORI_TYP(LCPDAT33), $APO = SAPO(LCPDAT33), $JERK = SJERK(LCPDAT33), $COLLMON_TOL_PRO[1] = USE_CM_PRO_VALUES(0)
          ;ENDFOLD
          ;FOLD SPTP P500 Vel=100 % PDAT19 Tool[1]:SMC Base[0] ;%{PE}
          ;FOLD Parameters ;%{h}
          ;Params IlfProvider=kukaroboter.basistech.inlineforms.movement.spline; Kuka.IsGlobalPoint=False; Kuka.PointName=P500; Kuka.BlendingEnabled=False; Kuka.MoveDataPtpName=PDAT19; Kuka.VelocityPtp=100; Kuka.VelocityFieldEnabled=True; Kuka.ColDetectFieldEnabled=True; Kuka.CurrentCDSetIndex=0; Kuka.MovementParameterFieldEnabled=True; IlfCommand=SPTP
          ;ENDFOLD
          SPTP XP500 WITH $VEL_AXIS[1] = SVEL_JOINT(100.0), $TOOL = STOOL2(FP500), $BASE = SBASE(FP500.BASE_NO), $IPO_MODE = SIPO_MODE(FP500.IPO_FRAME), $LOAD = SLOAD(FP500.TOOL_NO), $ACC_AXIS[1] = SACC_JOINT(PPDAT19), $APO = SAPO_PTP(PPDAT19), $GEAR_JERK[1] = SGEAR_JERK(PPDAT19), $COLLMON_TOL_PRO[1] = USE_CM_PRO_VALUES(0)
          ;ENDFOLD
          ;FOLD Gripper SET [1]Gripper1 State=[1]ABIERTA Wait 0.2[s] Check with Strategy 1 ;%{PE}
          ;FOLD Parameters Parameters ;%{h}
          ;Params IlfProvider=GripperTech.GripperSet;setgripper=1;setstate=1;setcont=nocont;waittime=0.2;errorstrategy=1
          ;ENDFOLD
          GRPg_SetStateAndCheck(1, 1, 0.2, 1)
          ;ENDFOLD
      ENDIF
      IF eatPosition == 51 THEN
          ;FOLD SPTP P151 Vel=100 % PDAT1 Tool[1]:SMC Base[0] ;%{PE}
          ;FOLD Parameters ;%{h}
          ;Params IlfProvider=kukaroboter.basistech.inlineforms.movement.spline; Kuka.IsGlobalPoint=False; Kuka.PointName=P151; Kuka.BlendingEnabled=False; Kuka.MoveDataPtpName=PDAT1; Kuka.VelocityPtp=100; Kuka.VelocityFieldEnabled=True; Kuka.ColDetectFieldEnabled=True; Kuka.CurrentCDSetIndex=0; Kuka.MovementParameterFieldEnabled=True; IlfCommand=SPTP
          ;ENDFOLD
          SPTP XP151 WITH $VEL_AXIS[1] = SVEL_JOINT(100.0), $TOOL = STOOL2(FP151), $BASE = SBASE(FP151.BASE_NO), $IPO_MODE = SIPO_MODE(FP151.IPO_FRAME), $LOAD = SLOAD(FP151.TOOL_NO), $ACC_AXIS[1] = SACC_JOINT(PPDAT1), $APO = SAPO_PTP(PPDAT1), $GEAR_JERK[1] = SGEAR_JERK(PPDAT1), $COLLMON_TOL_PRO[1] = USE_CM_PRO_VALUES(0)
          ;ENDFOLD
          ;FOLD SLIN P251 Vel=0.1 m/s CPDAT32 Tool[1]:SMC Base[0] ;%{PE}
          ;FOLD Parameters ;%{h}
          ;Params IlfProvider=kukaroboter.basistech.inlineforms.movement.spline; Kuka.IsGlobalPoint=False; Kuka.PointName=P251; Kuka.BlendingEnabled=False; Kuka.MoveDataName=CPDAT32; Kuka.VelocityPath=0.1; Kuka.VelocityFieldEnabled=True; Kuka.ColDetectFieldEnabled=True; Kuka.CurrentCDSetIndex=0; Kuka.MovementParameterFieldEnabled=True; IlfCommand=SLIN
          ;ENDFOLD
          SLIN XP251 WITH $VEL = SVEL_CP(0.1, , LCPDAT32), $TOOL = STOOL2(FP251), $BASE = SBASE(FP251.BASE_NO), $IPO_MODE = SIPO_MODE(FP251.IPO_FRAME), $LOAD = SLOAD(FP251.TOOL_NO), $ACC = SACC_CP(LCPDAT32), $ORI_TYPE = SORI_TYP(LCPDAT32), $APO = SAPO(LCPDAT32), $JERK = SJERK(LCPDAT32), $COLLMON_TOL_PRO[1] = USE_CM_PRO_VALUES(0)
          ;ENDFOLD
          ;FOLD Gripper SET [1]Gripper1 State=[2]CERRADA Wait 0.2[s] Check with Strategy 1 ;%{PE}
          ;FOLD Parameters Parameters ;%{h}
          ;Params IlfProvider=GripperTech.GripperSet;setgripper=1;setstate=2;setcont=nocont;waittime=0.2;errorstrategy=1
          ;ENDFOLD
          GRPg_SetStateAndCheck(1, 2, 0.2, 1)
          ;ENDFOLDinitialPosition
          ;FOLD SLIN P151 Vel=0.1 m/s CPDAT33 Tool[1]:SMC Base[0] ;%{PE}
          ;FOLD Parameters ;%{h}s
          ;Params IlfProvider=kukaroboter.basistech.inlineforms.movement.spline; Kuka.IsGlobalPoint=False; Kuka.PointName=P151; Kuka.BlendingEnabled=False; Kuka.MoveDataName=CPDAT33; Kuka.VelocityPath=0.1; Kuka.VelocityFieldEnabled=True; Kuka.ColDetectFieldEnabled=True; Kuka.CurrentCDSetIndex=0; Kuka.MovementParameterFieldEnabled=True; IlfCommand=SLIN
          ;ENDFOLD
          SLIN XP151 WITH $VEL = SVEL_CP(0.1, , LCPDAT33), $TOOL = STOOL2(FP151), $BASE = SBASE(FP151.BASE_NO), $IPO_MODE = SIPO_MODE(FP151.IPO_FRAME), $LOAD = SLOAD(FP151.TOOL_NO), $ACC = SACC_CP(LCPDAT33), $ORI_TYPE = SORI_TYP(LCPDAT33), $APO = SAPO(LCPDAT33), $JERK = SJERK(LCPDAT33), $COLLMON_TOL_PRO[1] = USE_CM_PRO_VALUES(0)
          ;ENDFOLD
          ;FOLD SPTP P500 Vel=100 % PDAT19 Tool[1]:SMC Base[0] ;%{PE}
          ;FOLD Parameters ;%{h}
          ;Params IlfProvider=kukaroboter.basistech.inlineforms.movement.spline; Kuka.IsGlobalPoint=False; Kuka.PointName=P500; Kuka.BlendingEnabled=False; Kuka.MoveDataPtpName=PDAT19; Kuka.VelocityPtp=100; Kuka.VelocityFieldEnabled=True; Kuka.ColDetectFieldEnabled=True; Kuka.CurrentCDSetIndex=0; Kuka.MovementParameterFieldEnabled=True; IlfCommand=SPTP
          ;ENDFOLD
          SPTP XP500 WITH $VEL_AXIS[1] = SVEL_JOINT(100.0), $TOOL = STOOL2(FP500), $BASE = SBASE(FP500.BASE_NO), $IPO_MODE = SIPO_MODE(FP500.IPO_FRAME), $LOAD = SLOAD(FP500.TOOL_NO), $ACC_AXIS[1] = SACC_JOINT(PPDAT19), $APO = SAPO_PTP(PPDAT19), $GEAR_JERK[1] = SGEAR_JERK(PPDAT19), $COLLMON_TOL_PRO[1] = USE_CM_PRO_VALUES(0)
          ;ENDFOLD
          ;FOLD Gripper SET [1]Gripper1 State=[1]ABIERTA Wait 0.2[s] Check with Strategy 1 ;%{PE}
          ;FOLD Parameters Parameters ;%{h}
          ;Params IlfProvider=GripperTech.GripperSet;setgripper=1;setstate=1;setcont=nocont;waittime=0.2;errorstrategy=1
          ;ENDFOLD
          GRPg_SetStateAndCheck(1, 1, 0.2, 1)
          ;ENDFOLD
      ENDIF
      IF eatPosition == 52 THEN
          ;FOLD SPTP P152 Vel=100 % PDAT1 Tool[1]:SMC Base[0] ;%{PE}
          ;FOLD Parameters ;%{h}
          ;Params IlfProvider=kukaroboter.basistech.inlineforms.movement.spline; Kuka.IsGlobalPoint=False; Kuka.PointName=P152; Kuka.BlendingEnabled=False; Kuka.MoveDataPtpName=PDAT1; Kuka.VelocityPtp=100; Kuka.VelocityFieldEnabled=True; Kuka.ColDetectFieldEnabled=True; Kuka.CurrentCDSetIndex=0; Kuka.MovementParameterFieldEnabled=True; IlfCommand=SPTP
          ;ENDFOLD
          SPTP XP152 WITH $VEL_AXIS[1] = SVEL_JOINT(100.0), $TOOL = STOOL2(FP152), $BASE = SBASE(FP152.BASE_NO), $IPO_MODE = SIPO_MODE(FP152.IPO_FRAME), $LOAD = SLOAD(FP152.TOOL_NO), $ACC_AXIS[1] = SACC_JOINT(PPDAT1), $APO = SAPO_PTP(PPDAT1), $GEAR_JERK[1] = SGEAR_JERK(PPDAT1), $COLLMON_TOL_PRO[1] = USE_CM_PRO_VALUES(0)
          ;ENDFOLD
          ;FOLD SLIN P252 Vel=0.1 m/s CPDAT32 Tool[1]:SMC Base[0] ;%{PE}
          ;FOLD Parameters ;%{h}
          ;Params IlfProvider=kukaroboter.basistech.inlineforms.movement.spline; Kuka.IsGlobalPoint=False; Kuka.PointName=P252; Kuka.BlendingEnabled=False; Kuka.MoveDataName=CPDAT32; Kuka.VelocityPath=0.1; Kuka.VelocityFieldEnabled=True; Kuka.ColDetectFieldEnabled=True; Kuka.CurrentCDSetIndex=0; Kuka.MovementParameterFieldEnabled=True; IlfCommand=SLIN
          ;ENDFOLD
          SLIN XP252 WITH $VEL = SVEL_CP(0.1, , LCPDAT32), $TOOL = STOOL2(FP252), $BASE = SBASE(FP252.BASE_NO), $IPO_MODE = SIPO_MODE(FP252.IPO_FRAME), $LOAD = SLOAD(FP252.TOOL_NO), $ACC = SACC_CP(LCPDAT32), $ORI_TYPE = SORI_TYP(LCPDAT32), $APO = SAPO(LCPDAT32), $JERK = SJERK(LCPDAT32), $COLLMON_TOL_PRO[1] = USE_CM_PRO_VALUES(0)
          ;ENDFOLD
          ;FOLD Gripper SET [1]Gripper1 State=[2]CERRADA Wait 0.2[s] Check with Strategy 1 ;%{PE}
          ;FOLD Parameters Parameters ;%{h}
          ;Params IlfProvider=GripperTech.GripperSet;setgripper=1;setstate=2;setcont=nocont;waittime=0.2;errorstrategy=1
          ;ENDFOLD
          GRPg_SetStateAndCheck(1, 2, 0.2, 1)
          ;ENDFOLDinitialPosition
          ;FOLD SLIN P152 Vel=0.1 m/s CPDAT33 Tool[1]:SMC Base[0] ;%{PE}
          ;FOLD Parameters ;%{h}s
          ;Params IlfProvider=kukaroboter.basistech.inlineforms.movement.spline; Kuka.IsGlobalPoint=False; Kuka.PointName=P152; Kuka.BlendingEnabled=False; Kuka.MoveDataName=CPDAT33; Kuka.VelocityPath=0.1; Kuka.VelocityFieldEnabled=True; Kuka.ColDetectFieldEnabled=True; Kuka.CurrentCDSetIndex=0; Kuka.MovementParameterFieldEnabled=True; IlfCommand=SLIN
          ;ENDFOLD
          SLIN XP152 WITH $VEL = SVEL_CP(0.1, , LCPDAT33), $TOOL = STOOL2(FP152), $BASE = SBASE(FP152.BASE_NO), $IPO_MODE = SIPO_MODE(FP152.IPO_FRAME), $LOAD = SLOAD(FP152.TOOL_NO), $ACC = SACC_CP(LCPDAT33), $ORI_TYPE = SORI_TYP(LCPDAT33), $APO = SAPO(LCPDAT33), $JERK = SJERK(LCPDAT33), $COLLMON_TOL_PRO[1] = USE_CM_PRO_VALUES(0)
          ;ENDFOLD
          ;FOLD SPTP P500 Vel=100 % PDAT19 Tool[1]:SMC Base[0] ;%{PE}
          ;FOLD Parameters ;%{h}
          ;Params IlfProvider=kukaroboter.basistech.inlineforms.movement.spline; Kuka.IsGlobalPoint=False; Kuka.PointName=P500; Kuka.BlendingEnabled=False; Kuka.MoveDataPtpName=PDAT19; Kuka.VelocityPtp=100; Kuka.VelocityFieldEnabled=True; Kuka.ColDetectFieldEnabled=True; Kuka.CurrentCDSetIndex=0; Kuka.MovementParameterFieldEnabled=True; IlfCommand=SPTP
          ;ENDFOLD
          SPTP XP500 WITH $VEL_AXIS[1] = SVEL_JOINT(100.0), $TOOL = STOOL2(FP500), $BASE = SBASE(FP500.BASE_NO), $IPO_MODE = SIPO_MODE(FP500.IPO_FRAME), $LOAD = SLOAD(FP500.TOOL_NO), $ACC_AXIS[1] = SACC_JOINT(PPDAT19), $APO = SAPO_PTP(PPDAT19), $GEAR_JERK[1] = SGEAR_JERK(PPDAT19), $COLLMON_TOL_PRO[1] = USE_CM_PRO_VALUES(0)
          ;ENDFOLD
          ;FOLD Gripper SET [1]Gripper1 State=[1]ABIERTA Wait 0.2[s] Check with Strategy 1 ;%{PE}
          ;FOLD Parameters Parameters ;%{h}
          ;Params IlfProvider=GripperTech.GripperSet;setgripper=1;setstate=1;setcont=nocont;waittime=0.2;errorstrategy=1
          ;ENDFOLD
          GRPg_SetStateAndCheck(1, 1, 0.2, 1)
          ;ENDFOLD
      ENDIF
      IF eatPosition == 53 THEN
          ;FOLD SPTP P153 Vel=100 % PDAT1 Tool[1]:SMC Base[0] ;%{PE}
          ;FOLD Parameters ;%{h}
          ;Params IlfProvider=kukaroboter.basistech.inlineforms.movement.spline; Kuka.IsGlobalPoint=False; Kuka.PointName=P153; Kuka.BlendingEnabled=False; Kuka.MoveDataPtpName=PDAT1; Kuka.VelocityPtp=100; Kuka.VelocityFieldEnabled=True; Kuka.ColDetectFieldEnabled=True; Kuka.CurrentCDSetIndex=0; Kuka.MovementParameterFieldEnabled=True; IlfCommand=SPTP
          ;ENDFOLD
          SPTP XP153 WITH $VEL_AXIS[1] = SVEL_JOINT(100.0), $TOOL = STOOL2(FP153), $BASE = SBASE(FP153.BASE_NO), $IPO_MODE = SIPO_MODE(FP153.IPO_FRAME), $LOAD = SLOAD(FP153.TOOL_NO), $ACC_AXIS[1] = SACC_JOINT(PPDAT1), $APO = SAPO_PTP(PPDAT1), $GEAR_JERK[1] = SGEAR_JERK(PPDAT1), $COLLMON_TOL_PRO[1] = USE_CM_PRO_VALUES(0)
          ;ENDFOLD
          ;FOLD SLIN P253 Vel=0.1 m/s CPDAT32 Tool[1]:SMC Base[0] ;%{PE}
          ;FOLD Parameters ;%{h}
          ;Params IlfProvider=kukaroboter.basistech.inlineforms.movement.spline; Kuka.IsGlobalPoint=False; Kuka.PointName=P253; Kuka.BlendingEnabled=False; Kuka.MoveDataName=CPDAT32; Kuka.VelocityPath=0.1; Kuka.VelocityFieldEnabled=True; Kuka.ColDetectFieldEnabled=True; Kuka.CurrentCDSetIndex=0; Kuka.MovementParameterFieldEnabled=True; IlfCommand=SLIN
          ;ENDFOLD
          SLIN XP253 WITH $VEL = SVEL_CP(0.1, , LCPDAT32), $TOOL = STOOL2(FP253), $BASE = SBASE(FP253.BASE_NO), $IPO_MODE = SIPO_MODE(FP253.IPO_FRAME), $LOAD = SLOAD(FP253.TOOL_NO), $ACC = SACC_CP(LCPDAT32), $ORI_TYPE = SORI_TYP(LCPDAT32), $APO = SAPO(LCPDAT32), $JERK = SJERK(LCPDAT32), $COLLMON_TOL_PRO[1] = USE_CM_PRO_VALUES(0)
          ;ENDFOLD
          ;FOLD Gripper SET [1]Gripper1 State=[2]CERRADA Wait 0.2[s] Check with Strategy 1 ;%{PE}
          ;FOLD Parameters Parameters ;%{h}
          ;Params IlfProvider=GripperTech.GripperSet;setgripper=1;setstate=2;setcont=nocont;waittime=0.2;errorstrategy=1
          ;ENDFOLD
          GRPg_SetStateAndCheck(1, 2, 0.2, 1)
          ;ENDFOLDinitialPosition
          ;FOLD SLIN P153 Vel=0.1 m/s CPDAT33 Tool[1]:SMC Base[0] ;%{PE}
          ;FOLD Parameters ;%{h}s
          ;Params IlfProvider=kukaroboter.basistech.inlineforms.movement.spline; Kuka.IsGlobalPoint=False; Kuka.PointName=P153; Kuka.BlendingEnabled=False; Kuka.MoveDataName=CPDAT33; Kuka.VelocityPath=0.1; Kuka.VelocityFieldEnabled=True; Kuka.ColDetectFieldEnabled=True; Kuka.CurrentCDSetIndex=0; Kuka.MovementParameterFieldEnabled=True; IlfCommand=SLIN
          ;ENDFOLD
          SLIN XP153 WITH $VEL = SVEL_CP(0.1, , LCPDAT33), $TOOL = STOOL2(FP153), $BASE = SBASE(FP153.BASE_NO), $IPO_MODE = SIPO_MODE(FP153.IPO_FRAME), $LOAD = SLOAD(FP153.TOOL_NO), $ACC = SACC_CP(LCPDAT33), $ORI_TYPE = SORI_TYP(LCPDAT33), $APO = SAPO(LCPDAT33), $JERK = SJERK(LCPDAT33), $COLLMON_TOL_PRO[1] = USE_CM_PRO_VALUES(0)
          ;ENDFOLD
          ;FOLD SPTP P500 Vel=100 % PDAT19 Tool[1]:SMC Base[0] ;%{PE}
          ;FOLD Parameters ;%{h}
          ;Params IlfProvider=kukaroboter.basistech.inlineforms.movement.spline; Kuka.IsGlobalPoint=False; Kuka.PointName=P500; Kuka.BlendingEnabled=False; Kuka.MoveDataPtpName=PDAT19; Kuka.VelocityPtp=100; Kuka.VelocityFieldEnabled=True; Kuka.ColDetectFieldEnabled=True; Kuka.CurrentCDSetIndex=0; Kuka.MovementParameterFieldEnabled=True; IlfCommand=SPTP
          ;ENDFOLD
          SPTP XP500 WITH $VEL_AXIS[1] = SVEL_JOINT(100.0), $TOOL = STOOL2(FP500), $BASE = SBASE(FP500.BASE_NO), $IPO_MODE = SIPO_MODE(FP500.IPO_FRAME), $LOAD = SLOAD(FP500.TOOL_NO), $ACC_AXIS[1] = SACC_JOINT(PPDAT19), $APO = SAPO_PTP(PPDAT19), $GEAR_JERK[1] = SGEAR_JERK(PPDAT19), $COLLMON_TOL_PRO[1] = USE_CM_PRO_VALUES(0)
          ;ENDFOLD
          ;FOLD Gripper SET [1]Gripper1 State=[1]ABIERTA Wait 0.2[s] Check with Strategy 1 ;%{PE}
          ;FOLD Parameters Parameters ;%{h}
          ;Params IlfProvider=GripperTech.GripperSet;setgripper=1;setstate=1;setcont=nocont;waittime=0.2;errorstrategy=1
          ;ENDFOLD
          GRPg_SetStateAndCheck(1, 1, 0.2, 1)
          ;ENDFOLD
      ENDIF
      IF eatPosition == 54 THEN
          ;FOLD SPTP P154 Vel=100 % PDAT1 Tool[1]:SMC Base[0] ;%{PE}
          ;FOLD Parameters ;%{h}
          ;Params IlfProvider=kukaroboter.basistech.inlineforms.movement.spline; Kuka.IsGlobalPoint=False; Kuka.PointName=P154; Kuka.BlendingEnabled=False; Kuka.MoveDataPtpName=PDAT1; Kuka.VelocityPtp=100; Kuka.VelocityFieldEnabled=True; Kuka.ColDetectFieldEnabled=True; Kuka.CurrentCDSetIndex=0; Kuka.MovementParameterFieldEnabled=True; IlfCommand=SPTP
          ;ENDFOLD
          SPTP XP154 WITH $VEL_AXIS[1] = SVEL_JOINT(100.0), $TOOL = STOOL2(FP154), $BASE = SBASE(FP154.BASE_NO), $IPO_MODE = SIPO_MODE(FP154.IPO_FRAME), $LOAD = SLOAD(FP154.TOOL_NO), $ACC_AXIS[1] = SACC_JOINT(PPDAT1), $APO = SAPO_PTP(PPDAT1), $GEAR_JERK[1] = SGEAR_JERK(PPDAT1), $COLLMON_TOL_PRO[1] = USE_CM_PRO_VALUES(0)
          ;ENDFOLD
          ;FOLD SLIN P254 Vel=0.1 m/s CPDAT32 Tool[1]:SMC Base[0] ;%{PE}
          ;FOLD Parameters ;%{h}
